C05497=1171.982,-20.083,-44.868,179.739,5.874,149.125
C05498=1171.976,-19.834,-44.881,179.742,5.874,149.124
C05499=1171.971,-19.584,-44.894,179.745,5.875,149.123
C05500=1171.966,-19.334,-44.907,179.746,5.875,149.123
C05501=1171.961,-19.085,-44.919,179.749,5.875,149.122
C05502=1171.956,-18.836,-44.932,179.751,5.876,149.122
C05503=1171.950,-18.586,-44.945,179.754,5.876,149.121
C05504=1171.946,-18.336,-44.958,179.756,5.877,149.120
C05505=1171.940,-18.086,-44.970,179.758,5.878,149.120
C05506=1171.935,-17.837,-44.983,179.761,5.878,149.119
C05507=1171.930,-17.588,-44.995,179.764,5.879,149.119
C05508=1171.925,-17.337,-45.009,179.766,5.879,149.118
C05509=1171.919,-17.088,-45.021,179.769,5.880,149.117
C05510=1171.914,-16.839,-45.034,179.771,5.880,149.117
C05511=1171.909,-16.589,-45.047,179.773,5.881,149.116
C05512=1171.904,-16.339,-45.060,179.776,5.882,149.116
C05513=1171.899,-16.090,-45.073,179.779,5.882,149.115
C05514=1171.894,-15.840,-45.085,179.781,5.883,149.114
C05515=1171.889,-15.590,-45.098,179.784,5.883,149.114
C05516=1171.883,-15.341,-45.112,179.785,5.883,149.113
C05517=1171.878,-15.091,-45.124,179.788,5.884,149.113
C05518=1171.874,-14.841,-45.137,179.791,5.884,149.112
C05519=1171.869,-14.592,-45.150,179.793,5.885,149.111
C05520=1171.863,-14.342,-45.163,179.795,5.886,149.111
C05521=1171.858,-14.092,-45.176,179.798,5.886,149.110
C05522=1171.853,-13.843,-45.189,179.800,5.887,149.110
C05523=1171.847,-13.593,-45.202,179.803,5.887,149.109
C05524=1171.842,-13.344,-45.214,179.806,5.888,149.108
C05525=1171.838,-13.094,-45.227,179.808,5.889,149.108
C05526=1171.832,-12.845,-45.240,179.810,5.889,149.107
C05527=1171.827,-12.595,-45.253,179.813,5.890,149.107
C05528=1171.822,-12.345,-45.266,179.815,5.890,149.106
C05529=1171.817,-12.096,-45.279,179.818,5.891,149.105
C05530=1171.812,-11.846,-45.293,179.820,5.892,149.105
C05531=1171.807,-11.597,-45.306,179.823,5.892,149.104
C05532=1171.801,-11.347,-45.319,179.825,5.892,149.103
C05533=1171.796,-11.097,-45.332,179.828,5.893,149.103
C05534=1171.791,-10.848,-45.344,179.830,5.894,149.102
C05535=1171.785,-10.598,-45.357,179.832,5.895,149.102
C05536=1171.781,-10.348,-45.370,179.835,5.895,149.101
C05537=1171.776,-10.099,-45.384,179.838,5.895,149.100
C05538=1171.771,-9.849,-45.397,179.840,5.896,149.100
C05539=1171.766,-9.600,-45.410,179.842,5.897,149.099
C05540=1171.760,-9.350,-45.423,179.845,5.897,149.098
C05541=1171.755,-9.100,-45.436,179.847,5.898,149.098
C05542=1171.750,-8.851,-45.449,179.850,5.898,149.097
C05543=1171.745,-8.601,-45.463,179.853,5.899,149.097
C05544=1171.740,-8.352,-45.476,179.855,5.900,149.096
C05545=1171.734,-8.102,-45.489,179.857,5.900,149.095
C05546=1171.730,-7.852,-45.502,179.860,5.901,149.095
C05547=1171.725,-7.604,-45.515,179.862,5.901,149.094
C05548=1171.720,-7.353,-45.529,179.864,5.901,149.094
C05549=1171.715,-7.104,-45.541,179.867,5.902,149.093
C05550=1171.709,-6.854,-45.554,179.869,5.902,149.092
C05551=1171.704,-6.605,-45.568,179.872,5.903,149.092
C05552=1171.699,-6.355,-45.581,179.874,5.904,149.091
C05553=1171.694,-6.105,-45.594,179.877,5.904,149.091
C05554=1171.689,-5.856,-45.608,179.879,5.905,149.090
C05555=1171.684,-5.606,-45.621,179.881,5.905,149.089
C05556=1171.678,-5.357,-45.634,179.884,5.906,149.089
C05557=1171.674,-5.106,-45.647,179.886,5.907,149.088
C05558=1171.668,-4.857,-45.661,179.889,5.907,149.088
C05559=1171.664,-4.607,-45.674,179.892,5.908,149.087
C05560=1171.658,-4.358,-45.687,179.894,5.908,149.086
C05561=1171.653,-4.109,-45.701,179.896,5.909,149.086
C05562=1171.648,-3.859,-45.714,179.900,5.910,149.085
C05563=1171.643,-3.610,-45.728,179.902,5.911,149.085
C05564=1171.638,-3.360,-45.741,179.905,5.911,149.084
C05565=1171.632,-3.110,-45.754,179.907,5.912,149.083
C05566=1171.627,-2.861,-45.768,179.909,5.913,149.083
C05567=1171.622,-2.611,-45.781,179.912,5.913,149.082
C05568=1171.617,-2.362,-45.795,179.914,5.914,149.082
C05569=1171.612,-2.112,-45.808,179.917,5.915,149.081
C05570=1171.607,-1.862,-45.821,179.920,5.915,149.080
C05571=1171.601,-1.613,-45.835,179.922,5.916,149.080
C05572=1171.597,-1.363,-45.848,179.924,5.916,149.079
C05573=1171.591,-1.114,-45.862,179.927,5.917,149.079
C05574=1171.586,-0.864,-45.875,179.929,5.918,149.078
C05575=1171.581,-0.615,-45.889,179.932,5.918,149.077
C05576=1171.576,-0.365,-45.902,179.934,5.919,149.077
C05577=1171.572,-0.115,-45.916,179.937,5.919,149.076
C05578=1171.566,0.134,-45.929,179.939,5.920,149.075
C05579=1171.561,0.384,-45.943,179.941,5.921,149.075
C05580=1171.556,0.633,-45.956,179.944,5.921,149.074
C05581=1171.551,0.883,-45.970,179.946,5.922,149.074
C05582=1171.545,1.133,-45.983,179.949,5.922,149.073
C05583=1171.541,1.382,-45.997,179.952,5.923,149.072
C05584=1171.535,1.632,-46.010,179.954,5.924,149.072
C05585=1171.530,1.901,-46.025,179.956,5.924,149.071
C05586=1171.524,2.171,-46.040,179.959,5.925,149.071
C05587=1171.519,2.440,-46.055,179.962,5.926,149.070
C05588=1171.513,2.708,-46.069,179.965,5.926,149.069
C05589=1171.508,2.959,-46.083,179.967,5.927,149.069
C05590=1171.503,3.208,-46.097,179.970,5.928,149.068
C05591=1171.498,3.458,-46.110,179.972,5.928,149.067
C05592=1171.493,3.707,-46.124,179.975,5.929,149.067
C05593=1171.488,3.956,-46.138,179.977,5.929,149.066
C05594=1171.483,4.206,-46.151,179.979,5.930,149.066
C05595=1171.478,4.456,-46.165,179.982,5.931,149.065
C05596=1171.473,4.705,-46.179,179.985,5.931,149.064
C05597=1171.467,4.956,-46.193,179.987,5.932,149.064
C05598=1171.462,5.204,-46.206,179.990,5.932,149.063
C05599=1171.457,5.454,-46.220,179.992,5.933,149.063
C05600=1171.452,5.704,-46.234,179.995,5.935,149.062
C05601=1171.447,5.953,-46.248,179.998,5.935,149.061
C05602=1171.442,6.203,-46.261,180.000,5.936,149.061
C05603=1171.437,6.453,-46.275,-179.998,5.936,149.060
C05604=1171.432,6.702,-46.289,-179.995,5.937,149.060
C05605=1171.427,6.952,-46.303,-179.993,5.938,149.059
C05606=1171.422,7.200,-46.317,-179.990,5.938,149.058
C05607=1171.417,7.451,-46.330,-179.988,5.939,149.058
C05608=1171.412,7.700,-46.344,-179.985,5.939,149.057
C05609=1171.406,7.949,-46.358,-179.983,5.940,149.057
C05610=1171.401,8.199,-46.373,-179.980,5.941,149.056
C05611=1171.397,8.449,-46.386,-179.978,5.941,149.055
C05612=1171.391,8.698,-46.399,-179.975,5.942,149.055
C05613=1171.386,8.948,-46.414,-179.973,5.942,149.054
C05614=1171.381,9.198,-46.428,-179.970,5.944,149.054
C05615=1171.376,9.447,-46.442,-179.968,5.945,149.053
C05616=1171.370,9.697,-46.455,-179.965,5.945,149.052
C05617=1171.365,9.947,-46.470,-179.962,5.946,149.052
C05618=1171.361,10.196,-46.483,-179.960,5.946,149.051
C05619=1171.356,10.445,-46.497,-179.957,5.947,149.051
C05620=1171.351,10.695,-46.512,-179.955,5.948,149.050
C05621=1171.346,10.945,-46.526,-179.953,5.948,149.049
C05622=1171.340,11.194,-46.539,-179.950,5.949,149.049
C05623=1171.335,11.444,-46.553,-179.948,5.949,149.048
C05624=1171.330,11.694,-46.568,-179.945,5.950,149.048
C05625=1171.325,11.943,-46.582,-179.942,5.951,149.047
C05626=1171.320,12.192,-46.595,-179.940,5.952,149.047
C05627=1171.315,12.442,-46.610,-179.937,5.953,149.046
C05628=1171.310,12.691,-46.624,-179.935,5.953,149.045
C05629=1171.305,12.941,-46.638,-179.932,5.954,149.045
C05630=1171.300,13.190,-46.652,-179.930,5.954,149.044
C05631=1171.295,13.440,-46.666,-179.927,5.955,149.044
C05632=1171.290,13.690,-46.681,-179.925,5.956,149.043
C05633=1171.285,13.939,-46.695,-179.923,5.956,149.042
C05634=1171.279,14.189,-46.708,-179.920,5.957,149.042
C05635=1171.274,14.439,-46.722,-179.917,5.958,149.041
C05636=1171.269,14.688,-46.737,-179.915,5.959,149.041
C05637=1171.264,14.938,-46.751,-179.912,5.960,149.040
C05638=1171.259,15.187,-46.765,-179.909,5.960,149.039
C05639=1171.254,15.437,-46.779,-179.907,5.961,149.039
C05640=1171.249,15.686,-46.793,-179.904,5.961,149.038
C05641=1171.244,15.936,-46.808,-179.902,5.962,149.038
C05642=1171.239,16.185,-46.823,-179.900,5.963,149.037
C05643=1171.233,16.434,-46.836,-179.896,5.964,149.036
C05644=1171.229,16.684,-46.851,-179.894,5.965,149.036
C05645=1171.224,16.934,-46.865,-179.892,5.965,149.035
C05646=1171.219,17.183,-46.879,-179.889,5.966,149.035
C05647=1171.214,17.433,-46.894,-179.887,5.967,149.034
C05648=1171.208,17.682,-46.908,-179.884,5.967,149.033
C05649=1171.203,17.932,-46.922,-179.882,5.968,149.033
C05650=1171.198,18.182,-46.936,-179.879,5.968,149.032
C05651=1171.193,18.431,-46.950,-179.877,5.970,149.032
C05652=1171.188,18.681,-46.965,-179.874,5.970,149.031
C05653=1171.184,18.930,-46.980,-179.871,5.971,149.030
C05654=1171.178,19.179,-46.994,-179.869,5.972,149.030
C05655=1171.173,19.429,-47.008,-179.866,5.972,149.029
C05656=1171.167,19.679,-47.023,-179.864,5.973,149.029
C05657=1171.162,19.928,-47.037,-179.862,5.974,149.028
C05658=1171.158,20.178,-47.051,-179.858,5.975,149.027
C05659=1171.153,20.427,-47.066,-179.856,5.976,149.027
C05660=1171.147,20.676,-47.080,-179.854,5.976,149.026
C05661=1171.142,20.926,-47.094,-179.851,5.977,149.026
C05662=1171.137,21.176,-47.109,-179.849,5.978,149.025
C05663=1171.132,21.425,-47.123,-179.846,5.978,149.024
C05664=1171.128,21.675,-47.138,-179.844,5.979,149.024
C05665=1171.122,21.925,-47.153,-179.841,5.980,149.023
C05666=1171.117,22.174,-47.167,-179.839,5.981,149.023
C05667=1171.112,22.424,-47.181,-179.836,5.981,149.022
C05668=1171.108,22.673,-47.196,-179.833,5.982,149.021
C05669=1171.102,22.922,-47.210,-179.831,5.983,149.021
C05670=1171.097,23.172,-47.225,-179.828,5.983,149.020
C05671=1171.091,23.422,-47.239,-179.826,5.985,149.020
C05672=1171.087,23.671,-47.254,-179.823,5.985,149.019
C05673=1171.082,23.921,-47.269,-179.820,5.986,149.019
C05674=1171.077,24.170,-47.283,-179.818,5.987,149.018
C05675=1171.072,24.419,-47.298,-179.816,5.987,149.017
C05676=1171.066,24.669,-47.313,-179.813,5.988,149.017
C05677=1171.062,24.919,-47.327,-179.810,5.989,149.016
C05678=1171.057,25.168,-47.342,-179.808,5.990,149.016
C05679=1171.052,25.418,-47.356,-179.805,5.991,149.015
C05680=1171.047,25.668,-47.371,-179.803,5.991,149.014
C05681=1171.042,25.917,-47.386,-179.801,5.992,149.014
C05682=1171.037,26.167,-47.401,-179.798,5.992,149.013
C05683=1171.032,26.416,-47.416,-179.795,5.994,149.013
C05684=1171.026,26.665,-47.429,-179.792,5.995,149.012
C05685=1171.021,26.915,-47.444,-179.790,5.995,149.012
C05686=1171.016,27.164,-47.459,-179.788,5.996,149.011
C05687=1171.011,27.414,-47.474,-179.785,5.996,149.010
C05688=1171.006,27.663,-47.489,-179.782,5.998,149.010
C05689=1171.001,27.932,-47.505,-179.780,5.999,149.009
C05690=1170.995,28.201,-47.521,-179.777,5.999,149.009
C05691=1170.990,28.470,-47.537,-179.774,6.000,149.008
C05692=1170.984,28.739,-47.553,-179.771,6.001,149.007
C05693=1170.980,28.988,-47.567,-179.769,6.002,149.007
C05694=1170.974,29.238,-47.582,-179.766,6.002,149.006
C05695=1170.969,29.487,-47.597,-179.764,6.004,149.006
C05696=1170.965,29.736,-47.612,-179.761,6.004,149.005
C05697=1170.959,29.986,-47.627,-179.758,6.005,149.004
C05698=1170.954,30.236,-47.642,-179.756,6.006,149.004
C05699=1170.949,30.486,-47.656,-179.753,6.006,149.003
C05700=1170.944,30.735,-47.671,-179.751,6.008,149.003
C05701=1170.939,30.984,-47.686,-179.748,6.008,149.002
C05702=1170.934,31.234,-47.701,-179.746,6.009,149.002
C05703=1170.929,31.483,-47.716,-179.743,6.010,149.001
C05704=1170.924,31.733,-47.731,-179.741,6.010,149.000
C05705=1170.919,31.982,-47.746,-179.738,6.012,149.000
C05706=1170.914,32.232,-47.761,-179.735,6.012,148.999
C05707=1170.909,32.482,-47.776,-179.733,6.013,148.999
C05708=1170.904,32.731,-47.791,-179.730,6.014,148.998
C05709=1170.899,32.981,-47.806,-179.728,6.015,148.998
C05710=1170.894,33.230,-47.821,-179.725,6.016,148.997
C05711=1170.889,33.480,-47.836,-179.722,6.016,148.996
C05712=1170.883,33.729,-47.851,-179.720,6.017,148.996
C05713=1170.879,33.978,-47.866,-179.718,6.018,148.995
C05714=1170.873,34.228,-47.881,-179.715,6.019,148.995
C05715=1170.868,34.477,-47.896,-179.712,6.020,148.994
C05716=1170.864,34.726,-47.911,-179.710,6.020,148.993
C05717=1170.858,34.976,-47.927,-179.707,6.021,148.993
C05718=1170.854,35.226,-47.941,-179.704,6.022,148.992
C05719=1170.849,35.476,-47.957,-179.702,6.023,148.992
C05720=1170.844,35.725,-47.972,-179.699,6.024,148.991
C05721=1170.838,35.975,-47.987,-179.697,6.025,148.991
C05722=1170.834,36.224,-48.002,-179.694,6.026,148.990
C05723=1170.828,36.473,-48.017,-179.691,6.026,148.989
C05724=1170.824,36.722,-48.032,-179.689,6.027,148.989
C05725=1170.818,36.972,-48.047,-179.687,6.028,148.988
C05726=1170.813,37.221,-48.062,-179.684,6.029,148.988
C05727=1170.809,37.472,-48.078,-179.681,6.030,148.987
C05728=1170.803,37.721,-48.094,-179.679,6.031,148.987
C05729=1170.798,37.970,-48.109,-179.676,6.031,148.986
C05730=1170.793,38.220,-48.124,-179.674,6.033,148.985
C05731=1170.788,38.469,-48.138,-179.671,6.033,148.985
C05732=1170.783,38.719,-48.154,-179.668,6.034,148.984
C05733=1170.779,38.968,-48.169,-179.666,6.035,148.984
C05734=1170.773,39.218,-48.185,-179.663,6.036,148.983
C05735=1170.768,39.467,-48.201,-179.661,6.037,148.982
C05736=1170.763,39.717,-48.215,-179.658,6.037,148.982
C05737=1170.758,39.966,-48.230,-179.656,6.038,148.981
C05738=1170.753,40.215,-48.245,-179.653,6.040,148.981
C05739=1170.748,40.465,-48.261,-179.650,6.040,148.980
C05740=1170.743,40.715,-48.277,-179.648,6.041,148.980
C05741=1170.738,40.964,-48.292,-179.645,6.041,148.979
C05742=1170.733,41.213,-48.308,-179.643,6.043,148.978
C05743=1170.728,41.462,-48.323,-179.640,6.044,148.978
C05744=1170.723,41.713,-48.339,-179.638,6.044,148.977
C05745=1170.718,41.962,-48.354,-179.635,6.045,148.977
C05746=1170.713,42.211,-48.369,-179.632,6.047,148.976
C05747=1170.708,42.460,-48.385,-179.630,6.047,148.976
C05748=1170.702,42.710,-48.400,-179.628,6.048,148.975
C05749=1170.698,42.960,-48.416,-179.624,6.049,148.974
C05750=1170.693,43.209,-48.431,-179.622,6.050,148.974
C05751=1170.688,43.458,-48.447,-179.620,6.051,148.973
C05752=1170.683,43.708,-48.462,-179.617,6.051,148.973
C05753=1170.678,43.958,-48.478,-179.614,6.053,148.972
C05754=1170.673,44.207,-48.493,-179.611,6.053,148.972
C05755=1170.667,44.456,-48.509,-179.609,6.054,148.971
C05756=1170.663,44.706,-48.524,-179.606,6.055,148.970
C05757=1170.658,44.956,-48.540,-179.604,6.056,148.970
C05758=1170.653,45.205,-48.555,-179.601,6.057,148.969
C05759=1170.648,45.454,-48.570,-179.599,6.057,148.969
C05760=1170.643,45.704,-48.586,-179.596,6.059,148.968
C05761=1170.638,45.954,-48.602,-179.593,6.059,148.968
C05762=1170.632,46.203,-48.618,-179.591,6.060,148.967
C05763=1170.628,46.452,-48.633,-179.588,6.062,148.966
C05764=1170.623,46.702,-48.649,-179.586,6.062,148.966
C05765=1170.618,46.951,-48.665,-179.583,6.063,148.965
C05766=1170.613,47.200,-48.680,-179.580,6.065,148.965
C05767=1170.608,47.450,-48.696,-179.578,6.065,148.964
C05768=1170.603,47.700,-48.711,-179.576,6.066,148.964
C05769=1170.598,47.949,-48.727,-179.572,6.067,148.963
C05770=1170.593,48.199,-48.743,-179.570,6.068,148.963
C05771=1170.588,48.448,-48.759,-179.568,6.069,148.962
C05772=1170.583,48.697,-48.774,-179.565,6.069,148.961
C05773=1170.578,48.947,-48.790,-179.562,6.071,148.961
C05774=1170.573,49.197,-48.806,-179.560,6.071,148.960
C05775=1170.568,49.446,-48.821,-179.557,6.072,148.960
C05776=1170.563,49.695,-48.838,-179.554,6.074,148.959
C05777=1170.558,49.945,-48.854,-179.552,6.074,148.959
C05778=1170.553,50.194,-48.869,-179.549,6.075,148.958
C05779=1170.548,50.444,-48.885,-179.547,6.077,148.958
C05780=1170.543,50.693,-48.901,-179.544,6.077,148.957
C05781=1170.538,50.942,-48.916,-179.542,6.078,148.956
C05782=1170.533,51.192,-48.932,-179.539,6.079,148.956
C05783=1170.528,51.441,-48.949,-179.536,6.080,148.955
C05784=1170.523,51.691,-48.965,-179.534,6.081,148.955
C05785=1170.518,51.941,-48.980,-179.531,6.082,148.954
C05786=1170.513,52.189,-48.996,-179.528,6.083,148.954
C05787=1170.509,52.439,-49.012,-179.526,6.084,148.953
C05788=1170.503,52.689,-49.028,-179.523,6.085,148.952
C05789=1170.499,52.938,-49.044,-179.520,6.085,148.952
C05790=1170.493,53.187,-49.060,-179.518,6.086,148.951
C05791=1170.488,53.437,-49.075,-179.515,6.088,148.951
C05792=1170.484,53.686,-49.092,-179.513,6.089,148.950
C05793=1170.478,53.955,-49.109,-179.510,6.090,148.950
C05794=1170.472,54.223,-49.126,-179.508,6.091,148.949
C05795=1170.467,54.492,-49.143,-179.504,6.092,148.948
C05796=1170.462,54.761,-49.160,-179.502,6.093,148.948
C05797=1170.457,55.010,-49.177,-179.499,6.094,148.947
C05798=1170.452,55.260,-49.193,-179.496,6.095,148.947
C05799=1170.447,55.509,-49.209,-179.494,6.096,148.946
C05800=1170.442,55.758,-49.225,-179.491,6.097,148.946
C05801=1170.437,56.008,-49.241,-179.489,6.098,148.945
C05802=1170.432,56.257,-49.257,-179.486,6.098,148.944
C05803=1170.427,56.506,-49.274,-179.483,6.100,148.944
C05804=1170.422,56.756,-49.289,-179.481,6.100,148.943
C05805=1170.417,57.005,-49.306,-179.478,6.101,148.943
C05806=1170.412,57.255,-49.321,-179.475,6.103,148.942
C05807=1170.408,57.504,-49.338,-179.473,6.103,148.942
C05808=1170.402,57.754,-49.354,-179.470,6.105,148.941
C05809=1170.398,58.003,-49.370,-179.467,6.105,148.940
C05810=1170.392,58.252,-49.386,-179.465,6.106,148.940
C05811=1170.387,58.502,-49.403,-179.462,6.108,148.939
C05812=1170.382,58.752,-49.419,-179.460,6.108,148.939
C05813=1170.377,59.001,-49.435,-179.457,6.109,148.938
C05814=1170.372,59.251,-49.451,-179.454,6.111,148.938
C05815=1170.367,59.500,-49.468,-179.452,6.111,148.937
C05816=1170.362,59.749,-49.484,-179.449,6.113,148.937
C05817=1170.357,59.999,-49.500,-179.446,6.113,148.936
C05818=1170.352,60.248,-49.516,-179.444,6.114,148.936
C05819=1170.348,60.497,-49.533,-179.441,6.115,148.935
C05820=1170.343,60.747,-49.548,-179.439,6.116,148.935
C05821=1170.337,60.996,-49.566,-179.436,6.118,148.934
C05822=1170.332,61.245,-49.582,-179.434,6.119,148.933
C05823=1170.327,61.495,-49.598,-179.431,6.119,148.933
C05824=1170.323,61.745,-49.615,-179.428,6.121,148.932
C05825=1170.318,61.994,-49.631,-179.426,6.122,148.932
C05826=1170.313,62.244,-49.647,-179.423,6.123,148.931
C05827=1170.307,62.493,-49.664,-179.421,6.124,148.931
C05828=1170.303,62.742,-49.681,-179.418,6.124,148.930
C05829=1170.297,62.992,-49.696,-179.415,6.126,148.930
C05830=1170.293,63.241,-49.713,-179.413,6.127,148.929
C05831=1170.288,63.490,-49.729,-179.410,6.128,148.929
C05832=1170.283,63.740,-49.746,-179.407,6.129,148.928
C05833=1170.278,63.990,-49.762,-179.405,6.130,148.928
C05834=1170.273,64.239,-49.779,-179.402,6.131,148.927
C05835=1170.268,64.488,-49.795,-179.400,6.132,148.926
C05836=1170.263,64.737,-49.812,-179.397,6.133,148.926
C05837=1170.258,64.987,-49.829,-179.394,6.134,148.925
C05838=1170.253,65.237,-49.845,-179.392,6.134,148.925
C05839=1170.248,65.486,-49.861,-179.389,6.136,148.924
C05840=1170.244,65.735,-49.878,-179.386,6.137,148.924
C05841=1170.238,65.985,-49.895,-179.384,6.138,148.923
C05842=1170.233,66.234,-49.911,-179.381,6.139,148.922
C05843=1170.229,66.483,-49.928,-179.378,6.141,148.922
C05844=1170.224,66.732,-49.944,-179.376,6.141,148.921
C05845=1170.218,66.982,-49.961,-179.374,6.142,148.921
C05846=1170.214,67.232,-49.978,-179.370,6.143,148.920
C05847=1170.209,67.481,-49.994,-179.368,6.144,148.920
C05848=1170.203,67.730,-50.011,-179.365,6.145,148.919
C05849=1170.199,67.980,-50.028,-179.363,6.146,148.919
C05850=1170.194,68.229,-50.044,-179.360,6.148,148.918
C05851=1170.189,68.478,-50.061,-179.357,6.149,148.918
C05852=1170.184,68.728,-50.078,-179.355,6.150,148.917
C05853=1170.179,68.977,-50.094,-179.352,6.151,148.917
C05854=1170.174,69.226,-50.112,-179.350,6.152,148.916
C05855=1170.169,69.476,-50.128,-179.347,6.153,148.915
C05856=1170.165,69.725,-50.145,-179.345,6.154,148.915
C05857=1170.159,69.975,-50.162,-179.341,6.155,148.914
C05858=1170.155,70.224,-50.178,-179.339,6.156,148.914
C05859=1170.150,70.473,-50.195,-179.336,6.157,148.913
C05860=1170.144,70.723,-50.212,-179.334,6.158,148.913
C05861=1170.140,70.972,-50.229,-179.331,6.160,148.912
C05862=1170.135,71.222,-50.246,-179.328,6.160,148.912
C05863=1170.130,71.471,-50.262,-179.326,6.162,148.911
C05864=1170.125,71.720,-50.279,-179.323,6.163,148.911
C05865=1170.120,71.970,-50.296,-179.321,6.164,148.910
C05866=1170.115,72.219,-50.313,-179.318,6.165,148.910
C05867=1170.110,72.468,-50.330,-179.316,6.166,148.909
C05868=1170.105,72.718,-50.346,-179.312,6.167,148.909
C05869=1170.100,72.968,-50.364,-179.310,6.168,148.908
C05870=1170.096,73.217,-50.381,-179.307,6.169,148.907
C05871=1170.090,73.466,-50.398,-179.305,6.170,148.907
C05872=1170.085,73.715,-50.415,-179.302,6.172,148.906
C05873=1170.080,73.965,-50.432,-179.299,6.172,148.906
C05874=1170.076,74.214,-50.449,-179.297,6.174,148.906
C05875=1170.070,74.464,-50.465,-179.294,6.175,148.905
C05876=1170.065,74.713,-50.482,-179.291,6.176,148.904
C05877=1170.060,74.962,-50.500,-179.289,6.177,148.904
C05878=1170.056,75.212,-50.517,-179.286,6.179,148.903
C05879=1170.051,75.462,-50.534,-179.283,6.179,148.903
C05880=1170.046,75.710,-50.550,-179.281,6.181,148.902
C05881=1170.041,75.959,-50.568,-179.278,6.181,148.902
C05882=1170.036,76.209,-50.585,-179.275,6.183,148.901
C05883=1170.031,76.459,-50.602,-179.273,6.184,148.901
C05884=1170.027,76.708,-50.619,-179.270,6.185,148.900
C05885=1170.021,76.957,-50.637,-179.268,6.186,148.900
C05886=1170.017,77.206,-50.653,-179.265,6.187,148.899
C05887=1170.011,77.456,-50.670,-179.262,6.188,148.899
C05888=1170.006,77.706,-50.688,-179.259,6.190,148.898
C05889=1170.002,77.955,-50.705,-179.257,6.190,148.897
C05890=1169.997,78.204,-50.722,-179.254,6.192,148.897
C05891=1169.992,78.453,-50.739,-179.252,6.193,148.896
C05892=1169.987,78.702,-50.757,-179.249,6.194,148.896
C05893=1169.982,78.952,-50.774,-179.246,6.195,148.895
C05894=1169.977,79.202,-50.791,-179.244,6.197,148.895
C05895=1169.972,79.451,-50.809,-179.241,6.197,148.894
C05896=1169.968,79.700,-50.825,-179.238,6.199,148.894
C05897=1169.962,79.969,-50.844,-179.236,6.199,148.893
C05898=1169.957,80.237,-50.863,-179.233,6.201,148.893
C05899=1169.951,80.506,-50.882,-179.230,6.202,148.892
C05900=1169.946,80.774,-50.899,-179.228,6.203,148.892
C05901=1169.941,81.023,-50.917,-179.224,6.205,148.891
C05902=1169.936,81.272,-50.935,-179.222,6.206,148.891
C05903=1169.931,81.522,-50.951,-179.219,6.207,148.890
C05904=1169.926,81.771,-50.969,-179.216,6.209,148.890
C05905=1169.921,82.021,-50.987,-179.214,6.209,148.889
C05906=1169.917,82.270,-51.004,-179.211,6.211,148.888
C05907=1169.912,82.520,-51.021,-179.209,6.212,148.888
C05908=1169.907,82.769,-51.039,-179.206,6.213,148.887
C05909=1169.902,83.019,-51.056,-179.203,6.214,148.887
C05910=1169.897,83.267,-51.074,-179.201,6.216,148.887
C05911=1169.892,83.517,-51.091,-179.198,6.216,148.886
C05912=1169.887,83.766,-51.109,-179.195,6.218,148.885
C05913=1169.882,84.015,-51.126,-179.193,6.218,148.885
C05914=1169.877,84.264,-51.143,-179.190,6.220,148.884
C05915=1169.873,84.514,-51.161,-179.187,6.221,148.884
C05916=1169.867,84.763,-51.179,-179.185,6.222,148.883
C05917=1169.862,85.013,-51.197,-179.182,6.224,148.883
C05918=1169.858,85.262,-51.213,-179.179,6.225,148.882
C05919=1169.853,85.511,-51.231,-179.177,6.226,148.882
C05920=1169.848,85.760,-51.249,-179.174,6.227,148.881
C05921=1169.843,86.010,-51.267,-179.171,6.228,148.881
C05922=1169.838,86.259,-51.284,-179.169,6.229,148.880
C05923=1169.833,86.509,-51.301,-179.166,6.231,148.880
C05924=1169.829,86.758,-51.319,-179.164,6.232,148.879
C05925=1169.824,87.007,-51.337,-179.161,6.233,148.879
C05926=1169.818,87.257,-51.354,-179.158,6.235,148.878
C05927=1169.814,87.506,-51.372,-179.156,6.235,148.878
C05928=1169.809,87.755,-51.390,-179.152,6.237,148.877
C05929=1169.804,88.005,-51.407,-179.150,6.238,148.877
C05930=1169.799,88.254,-51.425,-179.148,6.239,148.876
C05931=1169.794,88.503,-51.443,-179.145,6.240,148.876
C05932=1169.789,88.752,-51.461,-179.142,6.242,148.875
C05933=1169.784,89.002,-51.478,-179.139,6.243,148.875
C05934=1169.779,89.251,-51.496,-179.137,6.244,148.874
C05935=1169.774,89.500,-51.514,-179.134,6.246,148.874
C05936=1169.769,89.750,-51.532,-179.132,6.246,148.873
C05937=1169.764,89.999,-51.549,-179.129,6.248,148.873
C05938=1169.760,90.248,-51.567,-179.126,6.250,148.872
C05939=1169.755,90.497,-51.585,-179.123,6.250,148.872
C05940=1169.750,90.747,-51.603,-179.121,6.252,148.871
C05941=1169.745,90.996,-51.621,-179.118,6.252,148.870
C05942=1169.741,91.246,-51.638,-179.115,6.254,148.870
C05943=1169.736,91.495,-51.656,-179.113,6.255,148.870
C05944=1169.731,91.745,-51.674,-179.110,6.256,148.869
C05945=1169.726,91.994,-51.692,-179.107,6.258,148.869
C05946=1169.721,92.243,-51.710,-179.105,6.259,148.868
C05947=1169.716,92.492,-51.728,-179.102,6.260,148.868
C05948=1169.711,92.741,-51.746,-179.100,6.261,148.867
C05949=1169.706,92.991,-51.764,-179.097,6.263,148.867
C05950=1169.701,93.240,-51.782,-179.094,6.264,148.866
C05951=1169.696,93.490,-51.799,-179.092,6.265,148.866
C05952=1169.691,93.739,-51.817,-179.089,6.266,148.865
C05953=1169.687,93.989,-51.836,-179.086,6.267,148.865
C05954=1169.682,94.238,-51.854,-179.084,6.269,148.864
C05955=1169.677,94.487,-51.872,-179.081,6.270,148.864
C05956=1169.672,94.736,-51.890,-179.078,6.271,148.863
C05957=1169.667,94.985,-51.908,-179.076,6.273,148.863
C05958=1169.662,95.234,-51.926,-179.072,6.274,148.862
C05959=1169.658,95.484,-51.944,-179.070,6.275,148.862
C05960=1169.653,95.734,-51.962,-179.068,6.277,148.861
C05961=1169.648,95.983,-51.981,-179.065,6.277,148.861
C05962=1169.643,96.232,-51.999,-179.062,6.279,148.860
C05963=1169.638,96.481,-52.017,-179.060,6.281,148.860
C05964=1169.633,96.731,-52.035,-179.057,6.281,148.859
C05965=1169.628,96.980,-52.053,-179.054,6.283,148.859
C05966=1169.624,97.230,-52.071,-179.051,6.285,148.858
C05967=1169.619,97.479,-52.089,-179.049,6.285,148.858
C05968=1169.614,97.727,-52.108,-179.046,6.287,148.857
C05969=1169.609,97.976,-52.126,-179.044,6.288,148.857
C05970=1169.604,98.226,-52.144,-179.041,6.289,148.856
C05971=1169.599,98.475,-52.162,-179.038,6.291,148.856
C05972=1169.594,98.725,-52.180,-179.036,6.292,148.855
C05973=1169.589,98.974,-52.198,-179.033,6.293,148.855
C05974=1169.584,99.223,-52.216,-179.030,6.295,148.854
C05975=1169.580,99.473,-52.234,-179.028,6.296,148.854
C05976=1169.575,99.722,-52.254,-179.025,6.297,148.853
C05977=1169.570,99.971,-52.272,-179.022,6.299,148.853
C05978=1169.565,100.220,-52.290,-179.020,6.300,148.852
C05979=1169.560,100.470,-52.308,-179.017,6.301,148.852
C05980=1169.555,100.719,-52.326,-179.014,6.303,148.851
C05981=1169.550,100.968,-52.346,-179.012,6.304,148.851
C05982=1169.545,101.218,-52.364,-179.009,6.305,148.850
C05983=1169.541,101.467,-52.382,-179.006,6.307,148.850
C05984=1169.536,101.717,-52.400,-179.004,6.308,148.849
C05985=1169.532,101.965,-52.419,-179.001,6.309,148.849
C05986=1169.526,102.215,-52.437,-178.998,6.311,148.848
C05987=1169.521,102.464,-52.455,-178.996,6.312,148.848
C05988=1169.517,102.714,-52.474,-178.992,6.313,148.847
C05989=1169.511,102.963,-52.493,-178.990,6.315,148.847
C05990=1169.507,103.212,-52.511,-178.988,6.316,148.846
C05991=1169.502,103.461,-52.529,-178.985,6.317,148.846
C05992=1169.498,103.710,-52.548,-178.982,6.319,148.845
C05993=1169.492,103.960,-52.566,-178.980,6.320,148.845
C05994=1169.487,104.209,-52.584,-178.977,6.321,148.845
C05995=1169.483,104.458,-52.603,-178.974,6.323,148.844
C05996=1169.477,104.708,-52.622,-178.972,6.324,148.844
C05997=1169.473,104.956,-52.641,-178.969,6.325,148.843
C05998=1169.468,105.206,-52.659,-178.966,6.327,148.843
C05999=1169.463,105.456,-52.678,-178.963,6.328,148.842
C06000=1169.458,105.704,-52.696,-178.961,6.329,148.842
C06001=1169.452,105.973,-52.716,-178.958,6.331,148.841
C06002=1169.448,106.242,-52.736,-178.955,6.332,148.841
C06003=1169.442,106.510,-52.757,-178.952,6.334,148.840
C06004=1169.437,106.778,-52.776,-178.949,6.335,148.840
C06005=1169.433,107.027,-52.796,-178.947,6.336,148.839
C06006=1169.428,107.277,-52.814,-178.944,6.338,148.839
C06007=1169.423,107.525,-52.833,-178.941,6.339,148.838
C06008=1169.418,107.775,-52.851,-178.939,6.340,148.838
C06009=1169.413,108.024,-52.870,-178.936,6.342,148.837
C06010=1169.408,108.274,-52.889,-178.933,6.343,148.837
C06011=1169.404,108.523,-52.908,-178.930,6.345,148.836
C06012=1169.399,108.772,-52.926,-178.928,6.346,148.836
C06013=1169.394,109.021,-52.945,-178.925,6.347,148.835
C06014=1169.389,109.270,-52.963,-178.922,6.349,148.835
C06015=1169.384,109.519,-52.983,-178.920,6.350,148.834
C06016=1169.380,109.769,-53.001,-178.917,6.352,148.834
C06017=1169.374,110.018,-53.020,-178.914,6.353,148.833
C06018=1169.370,110.267,-53.039,-178.911,6.355,148.833
C06019=1169.365,110.517,-53.058,-178.909,6.356,148.833
C06020=1169.361,110.766,-53.077,-178.906,6.357,148.832
C06021=1169.355,111.015,-53.096,-178.903,6.359,148.832
C06022=1169.350,111.264,-53.114,-178.901,6.360,148.831
C06023=1169.346,111.514,-53.134,-178.898,6.361,148.831
C06024=1169.341,111.763,-53.152,-178.895,6.363,148.830
C06025=1169.336,112.012,-53.172,-178.892,6.365,148.830
C06026=1169.331,112.261,-53.190,-178.890,6.365,148.829
C06027=1169.327,112.511,-53.210,-178.888,6.367,148.829
C06028=1169.322,112.760,-53.228,-178.884,6.369,148.828
C06029=1169.317,113.009,-53.248,-178.882,6.370,148.828
C06030=1169.312,113.258,-53.267,-178.880,6.371,148.827
C06031=1169.307,113.507,-53.285,-178.877,6.373,148.827
C06032=1169.302,113.757,-53.305,-178.874,6.374,148.826
C06033=1169.297,114.005,-53.323,-178.871,6.376,148.826
C06034=1169.293,114.255,-53.343,-178.869,6.377,148.826
C06035=1169.287,114.505,-53.361,-178.866,6.379,148.825
C06036=1169.283,114.754,-53.381,-178.863,6.380,148.825
C06037=1169.278,115.003,-53.400,-178.860,6.382,148.824
C06038=1169.274,115.252,-53.419,-178.858,6.383,148.824
C06039=1169.268,115.501,-53.438,-178.855,6.384,148.823
C06040=1169.263,115.751,-53.457,-178.852,6.386,148.823
C06041=1169.259,116.000,-53.476,-178.849,6.387,148.822
C06042=1169.254,116.249,-53.495,-178.847,6.388,148.822
C06043=1169.248,116.498,-53.515,-178.845,6.390,148.821
C06044=1169.244,116.747,-53.534,-178.841,6.391,148.821
C06045=1169.240,116.997,-53.553,-178.839,6.393,148.820
C06046=1169.234,117.246,-53.573,-178.837,6.394,148.820
C06047=1169.230,117.495,-53.592,-178.834,6.396,148.820
C06048=1169.225,117.744,-53.610,-178.831,6.397,148.819
C06049=1169.220,117.994,-53.630,-178.828,6.399,148.819
C06050=1169.215,118.243,-53.649,-178.825,6.401,148.818
C06051=1169.211,118.492,-53.668,-178.823,6.401,148.818
C06052=1169.205,118.741,-53.688,-178.820,6.403,148.817
C06053=1169.201,118.991,-53.707,-178.817,6.405,148.817
C06054=1169.197,119.240,-53.726,-178.815,6.406,148.816
C06055=1169.191,119.489,-53.746,-178.812,6.407,148.816
C06056=1169.186,119.738,-53.765,-178.810,6.409,148.816
C06057=1169.181,119.987,-53.785,-178.807,6.410,148.815
C06058=1169.177,120.236,-53.804,-178.804,6.412,148.815
C06059=1169.172,120.486,-53.823,-178.801,6.414,148.814
C06060=1169.167,120.735,-53.843,-178.799,6.415,148.814
C06061=1169.162,120.984,-53.862,-178.796,6.416,148.813
C06062=1169.157,121.233,-53.882,-178.793,6.418,148.813
C06063=1169.153,121.482,-53.901,-178.790,6.419,148.812
C06064=1169.148,121.731,-53.921,-178.788,6.421,148.812
C06065=1169.143,121.980,-53.940,-178.786,6.422,148.811
C06066=1169.138,122.230,-53.960,-178.783,6.424,148.811
C06067=1169.134,122.479,-53.980,-178.780,6.425,148.810
C06068=1169.129,122.728,-53.998,-178.777,6.427,148.810
C06069=1169.124,122.978,-54.018,-178.774,6.429,148.810
C06070=1169.119,123.226,-54.037,-178.772,6.430,148.809
C06071=1169.114,123.476,-54.057,-178.769,6.431,148.809
C06072=1169.110,123.725,-54.077,-178.766,6.433,148.808
C06073=1169.104,123.974,-54.097,-178.763,6.434,148.808
C06074=1169.100,124.223,-54.116,-178.761,6.436,148.807
C06075=1169.096,124.473,-54.135,-178.759,6.437,148.807
C06076=1169.091,124.722,-54.155,-178.756,6.439,148.807
C06077=1169.086,124.970,-54.175,-178.753,6.440,148.806
C06078=1169.081,125.220,-54.195,-178.750,6.442,148.806
C06079=1169.076,125.470,-54.214,-178.747,6.444,148.805
C06080=1169.071,125.718,-54.234,-178.745,6.445,148.805
C06081=1169.067,125.967,-54.254,-178.742,6.446,148.804
C06082=1169.062,126.217,-54.274,-178.740,6.448,148.804
C06083=1169.057,126.466,-54.293,-178.737,6.449,148.803
C06084=1169.052,126.715,-54.313,-178.734,6.451,148.803
C06085=1169.047,126.964,-54.333,-178.731,6.453,148.803
C06086=1169.043,127.214,-54.353,-178.728,6.455,148.802
C06087=1169.037,127.463,-54.372,-178.726,6.455,148.802
C06088=1169.033,127.712,-54.392,-178.723,6.457,148.801
C06089=1169.028,127.961,-54.412,-178.720,6.459,148.801
C06090=1169.023,128.211,-54.432,-178.718,6.460,148.800
C06091=1169.018,128.459,-54.452,-178.715,6.462,148.800
C06092=1169.014,128.709,-54.471,-178.712,6.464,148.800
C06093=1169.009,128.958,-54.492,-178.710,6.466,148.799
C06094=1169.004,129.207,-54.511,-178.707,6.466,148.799
C06095=1168.999,129.456,-54.531,-178.704,6.468,148.798
C06096=1168.995,129.705,-54.551,-178.702,6.470,148.798
C06097=1168.990,129.955,-54.571,-178.699,6.471,148.797
C06098=1168.985,130.204,-54.591,-178.696,6.473,148.797
C06099=1168.980,130.452,-54.610,-178.693,6.475,148.797
C06100=1168.976,130.701,-54.631,-178.691,6.476,148.796
C06101=1168.971,130.951,-54.650,-178.688,6.477,148.796
C06102=1168.966,131.200,-54.671,-178.685,6.479,148.795
C06103=1168.962,131.449,-54.690,-178.683,6.480,148.795
C06104=1168.957,131.698,-54.710,-178.680,6.482,148.794
C06105=1168.951,131.967,-54.732,-178.677,6.484,148.794
C06106=1168.946,132.235,-54.753,-178.674,6.485,148.793
C06107=1168.941,132.504,-54.775,-178.671,6.487,148.793
C06108=1168.936,132.772,-54.797,-178.669,6.489,148.793
C06109=1168.931,133.022,-54.816,-178.666,6.491,148.792
C06110=1168.927,133.271,-54.837,-178.663,6.492,148.792
C06111=1168.921,133.520,-54.858,-178.660,6.494,148.791
C06112=1168.917,133.770,-54.877,-178.657,6.495,148.791
C06113=1168.912,134.019,-54.898,-178.655,6.497,148.790
C06114=1168.908,134.268,-54.917,-178.652,6.499,148.790
C06115=1168.903,134.516,-54.937,-178.649,6.501,148.790
C06116=1168.898,134.765,-54.958,-178.647,6.502,148.789
C06117=1168.893,135.015,-54.978,-178.645,6.503,148.789
C06118=1168.888,135.264,-54.998,-178.641,6.505,148.788
C06119=1168.884,135.513,-55.019,-178.639,6.506,148.788
C06120=1168.879,135.763,-55.038,-178.636,6.508,148.787
C06121=1168.874,136.012,-55.059,-178.633,6.510,148.787
C06122=1168.869,136.261,-55.080,-178.631,6.512,148.787
C06123=1168.865,136.510,-55.100,-178.628,6.513,148.786
C06124=1168.860,136.759,-55.119,-178.625,6.515,148.786
C06125=1168.854,137.008,-55.140,-178.622,6.517,148.786
C06126=1168.850,137.257,-55.161,-178.620,6.517,148.785
C06127=1168.845,137.507,-55.180,-178.617,6.519,148.785
C06128=1168.841,137.755,-55.201,-178.614,6.521,148.784
C06129=1168.836,138.005,-55.222,-178.612,6.523,148.784
C06130=1168.831,138.254,-55.242,-178.609,6.524,148.783
C06131=1168.827,138.503,-55.262,-178.606,6.526,148.783
C06132=1168.822,138.752,-55.282,-178.604,6.528,148.783
C06133=1168.817,139.001,-55.303,-178.601,6.530,148.782
C06134=1168.812,139.250,-55.323,-178.598,6.531,148.782
C06135=1168.808,139.499,-55.344,-178.596,6.533,148.781
C06136=1168.803,139.749,-55.365,-178.592,6.534,148.781
C06137=1168.798,139.998,-55.385,-178.590,6.536,148.780
C06138=1168.794,140.246,-55.405,-178.587,6.538,148.780
C06139=1168.788,140.496,-55.426,-178.585,6.539,148.780
C06140=1168.784,140.745,-55.446,-178.582,6.541,148.779
C06141=1168.779,140.995,-55.467,-178.579,6.542,148.779
C06142=1168.774,141.244,-55.487,-178.577,6.544,148.778
C06143=1168.770,141.492,-55.508,-178.574,6.546,148.778
C06144=1168.765,141.742,-55.529,-178.571,6.547,148.778
C06145=1168.760,141.991,-55.549,-178.569,6.549,148.777
C06146=1168.756,142.240,-55.569,-178.566,6.551,148.777
C06147=1168.751,142.489,-55.590,-178.563,6.553,148.777
C06148=1168.746,142.738,-55.611,-178.560,6.554,148.776
C06149=1168.741,142.987,-55.632,-178.557,6.556,148.776
C06150=1168.737,143.236,-55.652,-178.555,6.558,148.775
C06151=1168.732,143.485,-55.673,-178.552,6.559,148.775
C06152=1168.727,143.734,-55.693,-178.549,6.561,148.774
C06153=1168.722,143.984,-55.714,-178.547,6.563,148.774
C06154=1168.717,144.232,-55.735,-178.544,6.565,148.774
C06155=1168.713,144.481,-55.755,-178.541,6.566,148.773
C06156=1168.708,144.731,-55.776,-178.538,6.568,148.773
C06157=1168.703,144.980,-55.797,-178.536,6.570,148.772
C06158=1168.698,145.229,-55.817,-178.534,6.571,148.772
C06159=1168.694,145.477,-55.839,-178.531,6.572,148.772
C06160=1168.689,145.726,-55.860,-178.528,6.574,148.771
C06161=1168.684,145.975,-55.880,-178.526,6.576,148.771
C06162=1168.679,146.225,-55.901,-178.523,6.578,148.771
C06163=1168.675,146.474,-55.922,-178.520,6.579,148.770
C06164=1168.670,146.724,-55.943,-178.517,6.581,148.770
C06165=1168.665,146.973,-55.964,-178.514,6.583,148.769
C06166=1168.661,147.221,-55.985,-178.512,6.584,148.769
C06167=1168.656,147.470,-56.006,-178.509,6.586,148.768
C06168=1168.651,147.719,-56.026,-178.506,6.588,148.768
C06169=1168.646,147.969,-56.047,-178.503,6.590,148.768
C06170=1168.642,148.218,-56.067,-178.501,6.591,148.767
C06171=1168.637,148.466,-56.089,-178.498,6.593,148.767
C06172=1168.632,148.716,-56.110,-178.495,6.595,148.767
C06173=1168.628,148.965,-56.131,-178.493,6.596,148.766
C06174=1168.623,149.214,-56.152,-178.490,6.598,148.766
C06175=1168.618,149.463,-56.173,-178.487,6.600,148.765
C06176=1168.613,149.712,-56.194,-178.485,6.602,148.765
C06177=1168.608,149.961,-56.215,-178.482,6.603,148.765
C06178=1168.605,150.210,-56.236,-178.479,6.605,148.764
C06179=1168.600,150.460,-56.257,-178.476,6.607,148.764
C06180=1168.594,150.709,-56.278,-178.474,6.609,148.763
C06181=1168.590,150.957,-56.299,-178.471,6.610,148.763
C06182=1168.585,151.206,-56.320,-178.468,6.612,148.763
C06183=1168.580,151.456,-56.341,-178.466,6.614,148.762
C06184=1168.576,151.705,-56.363,-178.463,6.616,148.762
C06185=1168.571,151.954,-56.384,-178.460,6.617,148.762
C06186=1168.566,152.203,-56.405,-178.458,6.619,148.761
C06187=1168.561,152.452,-56.426,-178.455,6.621,148.761
C06188=1168.557,152.701,-56.447,-178.452,6.623,148.760
C06189=1168.552,152.950,-56.469,-178.450,6.624,148.760
C06190=1168.547,153.199,-56.490,-178.447,6.626,148.760
C06191=1168.542,153.448,-56.511,-178.444,6.628,148.759
C06192=1168.538,153.697,-56.532,-178.441,6.630,148.759
C06193=1168.533,153.946,-56.553,-178.439,6.631,148.759
C06194=1168.528,154.196,-56.575,-178.436,6.633,148.758
C06195=1168.524,154.444,-56.596,-178.433,6.635,148.758
C06196=1168.519,154.693,-56.617,-178.431,6.637,148.757
C06197=1168.514,154.942,-56.638,-178.427,6.639,148.757
C06198=1168.510,155.192,-56.660,-178.425,6.641,148.757
C06199=1168.505,155.440,-56.681,-178.422,6.643,148.756
C06200=1168.500,155.690,-56.702,-178.419,6.644,148.756
C06201=1168.495,155.939,-56.724,-178.417,6.646,148.756
C06202=1168.491,156.187,-56.745,-178.414,6.648,148.755
C06203=1168.486,156.437,-56.766,-178.411,6.650,148.755
C06204=1168.481,156.685,-56.788,-178.409,6.651,148.754
C06205=1168.477,156.935,-56.809,-178.406,6.653,148.754
C06206=1168.472,157.184,-56.831,-178.403,6.655,148.754
C06207=1168.467,157.432,-56.853,-178.400,6.657,148.753
C06208=1168.463,157.682,-56.874,-178.398,6.658,148.753
C06209=1168.457,157.950,-56.897,-178.395,6.660,148.753
C06210=1168.453,158.219,-56.920,-178.392,6.663,148.752
C06211=1168.447,158.489,-56.943,-178.389,6.665,148.752
C06212=1168.442,158.758,-56.966,-178.386,6.666,148.751
C06213=1168.438,159.007,-56.988,-178.384,6.668,148.751
C06214=1168.433,159.256,-57.010,-178.381,6.670,148.751
C06215=1168.428,159.504,-57.032,-178.378,6.672,148.750
C06216=1168.424,159.754,-57.053,-178.375,6.674,148.750
C06217=1168.419,160.003,-57.075,-178.372,6.676,148.750
C06218=1168.414,160.251,-57.096,-178.370,6.678,148.749
C06219=1168.410,160.501,-57.118,-178.367,6.679,148.749
C06220=1168.405,160.750,-57.139,-178.364,6.681,148.748
C06221=1168.400,160.999,-57.161,-178.362,6.683,148.748
C06222=1168.395,161.248,-57.183,-178.359,6.685,148.748
C06223=1168.391,161.497,-57.205,-178.356,6.686,148.747
C06224=1168.386,161.746,-57.227,-178.354,6.688,148.747
C06225=1168.381,161.995,-57.248,-178.351,6.690,148.747
C06226=1168.376,162.244,-57.269,-178.348,6.692,148.746
C06227=1168.372,162.493,-57.291,-178.345,6.693,148.746
C06228=1168.367,162.742,-57.313,-178.343,6.695,148.745
C06229=1168.363,162.991,-57.335,-178.340,6.698,148.745
C06230=1168.358,163.240,-57.357,-178.337,6.700,148.745
C06231=1168.353,163.489,-57.379,-178.335,6.702,148.745
C06232=1168.349,163.738,-57.401,-178.332,6.703,148.744
C06233=1168.344,163.987,-57.422,-178.329,6.705,148.744
C06234=1168.340,164.236,-57.444,-178.327,6.707,148.743
C06235=1168.335,164.485,-57.466,-178.324,6.709,148.743
C06236=1168.331,164.734,-57.488,-178.321,6.710,148.743
C06237=1168.326,164.982,-57.510,-178.318,6.712,148.742
C06238=1168.321,165.232,-57.532,-178.316,6.714,148.742
C06239=1168.316,165.481,-57.554,-178.313,6.716,148.742
C06240=1168.311,165.729,-57.576,-178.310,6.718,148.741
C06241=1168.307,165.979,-57.598,-178.307,6.720,148.741
C06242=1168.302,166.227,-57.619,-178.304,6.722,148.741
C06243=1168.298,166.477,-57.642,-178.302,6.724,148.740
C06244=1168.293,166.725,-57.663,-178.300,6.726,148.740
C06245=1168.288,166.975,-57.685,-178.297,6.727,148.740
C06246=1168.283,167.224,-57.708,-178.294,6.729,148.739
C06247=1168.279,167.473,-57.730,-178.291,6.732,148.739
C06248=1168.274,167.722,-57.751,-178.288,6.733,148.739
C06249=1168.269,167.971,-57.773,-178.286,6.735,148.738
C06250=1168.265,168.220,-57.795,-178.283,6.737,148.738
C06251=1168.260,168.469,-57.818,-178.280,6.739,148.737
C06252=1168.255,168.717,-57.840,-178.277,6.740,148.737
C06253=1168.251,168.967,-57.862,-178.275,6.742,148.737
C06254=1168.246,169.215,-57.884,-178.273,6.744,148.737
C06255=1168.241,169.465,-57.906,-178.269,6.747,148.736
C06256=1168.236,169.714,-57.928,-178.267,6.749,148.736
C06257=1168.232,169.962,-57.951,-178.264,6.750,148.735
C06258=1168.228,170.212,-57.973,-178.261,6.752,148.735
C06259=1168.222,170.461,-57.995,-178.259,6.754,148.735
C06260=1168.218,170.710,-58.017,-178.256,6.756,148.734
C06261=1168.213,170.959,-58.039,-178.254,6.758,148.734
C06262=1168.209,171.207,-58.062,-178.250,6.760,148.734
C06263=1168.203,171.456,-58.084,-178.248,6.762,148.734
C06264=1168.199,171.706,-58.106,-178.245,6.764,148.733
C06265=1168.195,171.954,-58.129,-178.242,6.766,148.733
C06266=1168.190,172.203,-58.151,-178.240,6.767,148.732
C06267=1168.185,172.453,-58.173,-178.237,6.769,148.732
C06268=1168.181,172.701,-58.195,-178.234,6.772,148.732
C06269=1168.176,172.950,-58.218,-178.232,6.774,148.732
C06270=1168.171,173.200,-58.240,-178.229,6.776,148.731
C06271=1168.167,173.448,-58.263,-178.226,6.777,148.731
C06272=1168.162,173.697,-58.285,-178.223,6.779,148.730
C06273=1168.157,173.946,-58.307,-178.221,6.781,148.730
C06274=1168.152,174.195,-58.330,-178.217,6.783,148.730
C06275=1168.148,174.444,-58.352,-178.215,6.785,148.730
C06276=1168.144,174.692,-58.375,-178.213,6.787,148.729
C06277=1168.139,174.942,-58.397,-178.210,6.789,148.729
C06278=1168.135,175.191,-58.420,-178.207,6.791,148.729
C06279=1168.129,175.440,-58.442,-178.205,6.793,148.728
C06280=1168.125,175.689,-58.464,-178.201,6.795,148.728
C06281=1168.121,175.938,-58.487,-178.199,6.797,148.727
C06282=1168.115,176.187,-58.509,-178.196,6.799,148.727
C06283=1168.111,176.435,-58.532,-178.194,6.801,148.727
C06284=1168.106,176.685,-58.555,-178.191,6.803,148.727
C06285=1168.102,176.933,-58.577,-178.188,6.805,148.726
C06286=1168.097,177.182,-58.601,-178.185,6.807,148.726
C06287=1168.093,177.431,-58.623,-178.182,6.809,148.726
C06288=1168.087,177.680,-58.646,-178.180,6.811,148.725
C06289=1168.083,177.929,-58.668,-178.178,6.812,148.725
C06290=1168.078,178.178,-58.691,-178.174,6.815,148.725
C06291=1168.073,178.427,-58.713,-178.172,6.817,148.724
C06292=1168.069,178.676,-58.736,-178.169,6.819,148.724
C06293=1168.065,178.925,-58.759,-178.167,6.821,148.724
C06294=1168.060,179.174,-58.782,-178.164,6.822,148.723
C06295=1168.055,179.422,-58.804,-178.161,6.825,148.723
C06296=1168.051,179.671,-58.827,-178.158,6.827,148.723
C06297=1168.046,179.921,-58.849,-178.155,6.829,148.722
C06298=1168.042,180.170,-58.873,-178.153,6.831,148.722
C06299=1168.037,180.418,-58.895,-178.150,6.833,148.722
C06300=1168.032,180.667,-58.918,-178.147,6.835,148.722
C06301=1168.027,180.916,-58.941,-178.145,6.837,148.721
C06302=1168.023,181.165,-58.964,-178.142,6.839,148.721
C06303=1168.018,181.413,-58.987,-178.140,6.841,148.721
C06304=1168.014,181.663,-59.009,-178.136,6.843,148.720
C06305=1168.009,181.912,-59.032,-178.134,6.845,148.720
C06306=1168.004,182.161,-59.056,-178.131,6.847,148.720
C06307=1168.000,182.410,-59.078,-178.128,6.849,148.719
C06308=1167.995,182.658,-59.101,-178.126,6.851,148.719
C06309=1167.990,182.907,-59.124,-178.123,6.853,148.719
C06310=1167.986,183.156,-59.147,-178.120,6.855,148.718
C06311=1167.981,183.405,-59.170,-178.118,6.857,148.718
C06312=1167.977,183.654,-59.194,-178.114,6.859,148.718
C06313=1167.972,183.924,-59.218,-178.112,6.861,148.718
C06314=1167.967,184.193,-59.243,-178.109,6.864,148.717
C06315=1167.962,184.463,-59.268,-178.106,6.866,148.717
C06316=1167.957,184.733,-59.292,-178.103,6.868,148.717
C06317=1167.952,184.982,-59.316,-178.100,6.870,148.716
C06318=1167.947,185.230,-59.339,-178.098,6.872,148.716
C06319=1167.943,185.479,-59.362,-178.095,6.874,148.716
C06320=1167.938,185.728,-59.385,-178.092,6.877,148.715
C06321=1167.934,185.977,-59.408,-178.089,6.878,148.715
C06322=1167.929,186.226,-59.432,-178.087,6.880,148.715
C06323=1167.925,186.475,-59.454,-178.084,6.882,148.714
C06324=1167.920,186.724,-59.478,-178.081,6.885,148.714
C06325=1167.916,186.973,-59.501,-178.079,6.887,148.714
C06326=1167.910,187.221,-59.524,-178.076,6.888,148.713
C06327=1167.906,187.470,-59.547,-178.073,6.890,148.713
C06328=1167.902,187.719,-59.570,-178.070,6.893,148.713
C06329=1167.897,187.968,-59.594,-178.068,6.895,148.713
C06330=1167.892,188.217,-59.617,-178.065,6.897,148.712
C06331=1167.887,188.466,-59.640,-178.062,6.900,148.712
C06332=1167.883,188.715,-59.664,-178.060,6.901,148.712
C06333=1167.878,188.964,-59.687,-178.057,6.903,148.711
C06334=1167.874,189.213,-59.710,-178.054,6.905,148.711
C06335=1167.869,189.462,-59.733,-178.051,6.908,148.711
C06336=1167.865,189.710,-59.757,-178.049,6.910,148.711
C06337=1167.860,189.958,-59.780,-178.046,6.911,148.710
C06338=1167.855,190.207,-59.804,-178.043,6.914,148.710
C06339=1167.850,190.456,-59.827,-178.041,6.916,148.710
C06340=1167.846,190.706,-59.850,-178.038,6.918,148.709
C06341=1167.841,190.955,-59.874,-178.035,6.920,148.709
C06342=1167.837,191.203,-59.898,-178.033,6.923,148.709
C06343=1167.833,191.452,-59.921,-178.030,6.924,148.709
C06344=1167.828,191.701,-59.944,-178.027,6.926,148.708
C06345=1167.823,191.950,-59.967,-178.024,6.929,148.708
C06346=1167.819,192.198,-59.991,-178.022,6.931,148.708
C06347=1167.814,192.447,-60.015,-178.019,6.933,148.707
C06348=1167.809,192.696,-60.038,-178.016,6.935,148.707
C06349=1167.805,192.945,-60.061,-178.014,6.937,148.707
C06350=1167.800,193.194,-60.085,-178.011,6.939,148.707
C06351=1167.796,193.443,-60.109,-178.008,6.941,148.706
C06352=1167.791,193.692,-60.132,-178.005,6.943,148.706
C06353=1167.786,193.940,-60.156,-178.003,6.945,148.706
C06354=1167.782,194.189,-60.180,-178.000,6.947,148.706
C06355=1167.777,194.438,-60.203,-177.997,6.950,148.705
C06356=1167.773,194.687,-60.227,-177.995,6.952,148.705
C06357=1167.768,194.936,-60.250,-177.992,6.954,148.705
C06358=1167.763,195.185,-60.274,-177.989,6.956,148.704
C06359=1167.759,195.433,-60.298,-177.987,6.958,148.704
C06360=1167.754,195.682,-60.321,-177.984,6.960,148.704
C06361=1167.750,195.931,-60.345,-177.981,6.963,148.704
C06362=1167.745,196.181,-60.370,-177.978,6.965,148.703
C06363=1167.741,196.429,-60.394,-177.976,6.967,148.703
C06364=1167.736,196.678,-60.417,-177.972,6.969,148.703
C06365=1167.731,196.927,-60.440,-177.970,6.971,148.703
C06366=1167.727,197.175,-60.464,-177.968,6.973,148.702
C06367=1167.722,197.425,-60.488,-177.964,6.976,148.702
C06368=1167.718,197.673,-60.512,-177.962,6.978,148.702
C06369=1167.713,197.922,-60.535,-177.959,6.980,148.701
C06370=1167.709,198.170,-60.559,-177.956,6.982,148.701
C06371=1167.703,198.419,-60.584,-177.954,6.984,148.701
C06372=1167.699,198.668,-60.607,-177.951,6.986,148.701
C06373=1167.695,198.917,-60.632,-177.948,6.989,148.700
C06374=1167.690,199.166,-60.655,-177.946,6.991,148.700
C06375=1167.686,199.415,-60.679,-177.943,6.993,148.700
C06376=1167.681,199.664,-60.703,-177.940,6.995,148.700
C06377=1167.676,199.912,-60.727,-177.938,6.997,148.699
C06378=1167.672,200.161,-60.751,-177.935,7.000,148.699
C06379=1167.667,200.410,-60.775,-177.932,7.002,148.699
C06380=1167.663,200.659,-60.799,-177.930,7.004,148.699
C06381=1167.659,200.907,-60.823,-177.926,7.006,148.698
C06382=1167.653,201.157,-60.847,-177.924,7.009,148.698
C06383=1167.649,201.405,-60.871,-177.922,7.010,148.698
C06384=1167.645,201.654,-60.895,-177.918,7.013,148.698
C06385=1167.640,201.903,-60.919,-177.916,7.015,148.697
C06386=1167.635,202.152,-60.944,-177.913,7.018,148.697
C06387=1167.631,202.400,-60.968,-177.910,7.019,148.697
C06388=1167.626,202.649,-60.992,-177.908,7.022,148.697
C06389=1167.622,202.898,-61.015,-177.905,7.024,148.696
C06390=1167.617,203.147,-61.040,-177.902,7.026,148.696
C06391=1167.613,203.396,-61.064,-177.900,7.028,148.696
C06392=1167.608,203.644,-61.088,-177.897,7.031,148.695
C06393=1167.603,203.893,-61.113,-177.894,7.033,148.695
C06394=1167.599,204.142,-61.136,-177.891,7.035,148.695
C06395=1167.595,204.391,-61.161,-177.888,7.037,148.695
C06396=1167.590,204.640,-61.186,-177.886,7.039,148.695
C06397=1167.585,204.888,-61.210,-177.883,7.042,148.694
C06398=1167.581,205.137,-61.234,-177.881,7.044,148.694
C06399=1167.576,205.385,-61.258,-177.878,7.047,148.694
C06400=1167.572,205.634,-61.283,-177.875,7.048,148.693
C06401=1167.567,205.883,-61.306,-177.873,7.050,148.693
C06402=1167.562,206.132,-61.331,-177.869,7.053,148.693
C06403=1167.558,206.381,-61.355,-177.867,7.055,148.693
C06404=1167.553,206.630,-61.380,-177.864,7.058,148.693
C06405=1167.549,206.878,-61.404,-177.862,7.060,148.692
C06406=1167.544,207.127,-61.429,-177.859,7.062,148.692
C06407=1167.540,207.376,-61.453,-177.856,7.064,148.692
C06408=1167.536,207.625,-61.477,-177.854,7.066,148.692
C06409=1167.530,207.873,-61.502,-177.850,7.069,148.691
C06410=1167.527,208.123,-61.526,-177.848,7.071,148.691
C06411=1167.521,208.371,-61.551,-177.846,7.073,148.691
C06412=1167.517,208.620,-61.575,-177.842,7.075,148.691
C06413=1167.512,208.868,-61.600,-177.840,7.078,148.690
C06414=1167.508,209.117,-61.624,-177.837,7.080,148.690
C06415=1167.503,209.366,-61.649,-177.835,7.082,148.690
C06416=1167.499,209.615,-61.673,-177.831,7.085,148.690
C06417=1167.494,209.885,-61.700,-177.829,7.087,148.689
C06418=1167.489,210.156,-61.727,-177.826,7.090,148.689
C06419=1167.484,210.427,-61.754,-177.823,7.092,148.689
C06420=1167.479,210.697,-61.780,-177.820,7.095,148.689
C06421=1167.474,210.945,-61.805,-177.817,7.097,148.689
C06422=1167.470,211.195,-61.830,-177.815,7.099,148.688
C06423=1167.465,211.443,-61.855,-177.812,7.102,148.688
C06424=1167.461,211.691,-61.879,-177.809,7.103,148.688
C06425=1167.457,211.940,-61.904,-177.806,7.106,148.688
C06426=1167.451,212.189,-61.929,-177.804,7.108,148.687
C06427=1167.448,212.438,-61.953,-177.801,7.111,148.687
C06428=1167.443,212.686,-61.979,-177.798,7.113,148.687
C06429=1167.438,212.935,-62.003,-177.796,7.116,148.687
C06430=1167.434,213.184,-62.028,-177.793,7.118,148.686
C06431=1167.429,213.433,-62.052,-177.790,7.119,148.686
C06432=1167.425,213.681,-62.077,-177.787,7.122,148.686
C06433=1167.420,213.930,-62.102,-177.785,7.124,148.686
C06434=1167.415,214.179,-62.127,-177.782,7.127,148.686
C06435=1167.412,214.427,-62.152,-177.779,7.129,148.685
C06436=1167.406,214.676,-62.177,-177.777,7.132,148.685
C06437=1167.402,214.926,-62.202,-177.774,7.134,148.685
C06438=1167.398,215.173,-62.226,-177.771,7.137,148.685
C06439=1167.393,215.423,-62.252,-177.769,7.138,148.684
C06440=1167.388,215.671,-62.276,-177.766,7.141,148.684
C06441=1167.385,215.920,-62.301,-177.763,7.143,148.684
C06442=1167.379,216.169,-62.326,-177.760,7.146,148.684
C06443=1167.375,216.417,-62.351,-177.758,7.148,148.684
C06444=1167.371,216.666,-62.376,-177.755,7.151,148.683
C06445=1167.366,216.915,-62.401,-177.752,7.152,148.683
C06446=1167.361,217.163,-62.426,-177.749,7.155,148.683
C06447=1167.356,217.412,-62.451,-177.747,7.157,148.683
C06448=1167.353,217.661,-62.476,-177.744,7.160,148.683
C06449=1167.348,217.909,-62.501,-177.741,7.162,148.682
C06450=1167.344,218.158,-62.527,-177.739,7.165,148.682
C06451=1167.338,218.407,-62.551,-177.736,7.167,148.682
C06452=1167.334,218.656,-62.577,-177.734,7.169,148.682
C06453=1167.330,218.905,-62.601,-177.730,7.171,148.681
C06454=1167.326,219.153,-62.627,-177.728,7.174,148.681
C06455=1167.321,219.402,-62.653,-177.725,7.176,148.681
C06456=1167.316,219.650,-62.677,-177.722,7.179,148.681
C06457=1167.312,219.899,-62.703,-177.720,7.181,148.681
C06458=1167.307,220.148,-62.728,-177.717,7.184,148.680
C06459=1167.303,220.396,-62.753,-177.714,7.186,148.680
C06460=1167.299,220.645,-62.778,-177.711,7.189,148.680
C06461=1167.294,220.894,-62.803,-177.709,7.191,148.680
C06462=1167.290,221.143,-62.829,-177.706,7.193,148.680
C06463=1167.285,221.391,-62.854,-177.704,7.195,148.679
C06464=1167.280,221.640,-62.879,-177.701,7.198,148.679
C06465=1167.276,221.888,-62.905,-177.698,7.200,148.679
C06466=1167.271,222.137,-62.930,-177.695,7.203,148.679
C06467=1167.267,222.386,-62.955,-177.693,7.205,148.679
C06468=1167.263,222.634,-62.980,-177.690,7.207,148.678
C06469=1167.259,222.883,-63.006,-177.687,7.210,148.678
C06470=1167.254,223.131,-63.031,-177.684,7.212,148.678
C06471=1167.249,223.381,-63.056,-177.682,7.214,148.678
C06472=1167.244,223.629,-63.082,-177.679,7.217,148.678
C06473=1167.240,223.878,-63.108,-177.677,7.219,148.677
C06474=1167.236,224.127,-63.133,-177.674,7.222,148.677
C06475=1167.231,224.375,-63.159,-177.671,7.224,148.677
C06476=1167.227,224.624,-63.184,-177.668,7.227,148.677
C06477=1167.222,224.873,-63.210,-177.665,7.229,148.677
C06478=1167.217,225.121,-63.235,-177.663,7.231,148.676
C06479=1167.213,225.370,-63.261,-177.660,7.234,148.676
C06480=1167.209,225.619,-63.286,-177.658,7.236,148.676
C06481=1167.204,225.867,-63.312,-177.655,7.239,148.676
C06482=1167.200,226.115,-63.338,-177.652,7.241,148.676
C06483=1167.196,226.364,-63.363,-177.649,7.244,148.676
C06484=1167.191,226.613,-63.388,-177.647,7.246,148.675
C06485=1167.186,226.862,-63.414,-177.644,7.249,148.675
C06486=1167.181,227.111,-63.440,-177.641,7.252,148.675
C06487=1167.177,227.359,-63.465,-177.639,7.253,148.675
C06488=1167.172,227.608,-63.491,-177.636,7.256,148.675
C06489=1167.168,227.857,-63.517,-177.633,7.258,148.674
C06490=1167.163,228.105,-63.542,-177.630,7.261,148.674
C06491=1167.159,228.354,-63.568,-177.628,7.263,148.674
C06492=1167.155,228.602,-63.594,-177.625,7.266,148.674
C06493=1167.151,228.851,-63.620,-177.622,7.269,148.674
C06494=1167.146,229.099,-63.645,-177.619,7.271,148.673
C06495=1167.141,229.348,-63.671,-177.617,7.273,148.673
C06496=1167.137,229.597,-63.698,-177.615,7.276,148.673
C06497=1167.133,229.845,-63.724,-177.611,7.278,148.673
C06498=1167.128,230.093,-63.749,-177.609,7.280,148.673
C06499=1167.124,230.342,-63.775,-177.606,7.283,148.673
C06500=1167.119,230.591,-63.800,-177.603,7.286,148.672
C06501=1167.114,230.840,-63.827,-177.601,7.288,148.672
C06502=1167.110,231.088,-63.852,-177.598,7.291,148.672
C06503=1167.105,231.337,-63.878,-177.595,7.293,148.672
C06504=1167.102,231.585,-63.904,-177.593,7.296,148.672
C06505=1167.097,231.834,-63.931,-177.589,7.298,148.672
C06506=1167.092,232.083,-63.956,-177.587,7.300,148.671
C06507=1167.088,232.331,-63.982,-177.585,7.303,148.671
C06508=1167.083,232.580,-64.008,-177.582,7.305,148.671
C06509=1167.079,232.829,-64.035,-177.579,7.308,148.671
C06510=1167.074,233.077,-64.060,-177.576,7.311,148.671
C06511=1167.070,233.326,-64.086,-177.574,7.313,148.671
C06512=1167.065,233.574,-64.112,-177.571,7.316,148.670
C06513=1167.061,233.823,-64.139,-177.569,7.318,148.670
C06514=1167.056,234.072,-64.164,-177.566,7.321,148.670
C06515=1167.052,234.320,-64.190,-177.563,7.324,148.670
C06516=1167.048,234.569,-64.217,-177.561,7.326,148.670
C06517=1167.043,234.818,-64.243,-177.557,7.328,148.670
C06518=1167.039,235.066,-64.268,-177.555,7.331,148.670
C06519=1167.034,235.314,-64.295,-177.552,7.333,148.669
C06520=1167.030,235.563,-64.321,-177.549,7.336,148.669
C06521=1167.025,235.834,-64.350,-177.546,7.339,148.669
C06522=1167.020,236.107,-64.379,-177.543,7.342,148.669
C06523=1167.015,236.378,-64.407,-177.540,7.344,148.669
C06524=1167.010,236.650,-64.436,-177.537,7.347,148.668
C06525=1167.006,236.898,-64.462,-177.535,7.349,148.668
C06526=1167.001,237.147,-64.489,-177.532,7.352,148.668
C06527=1166.997,237.396,-64.515,-177.529,7.355,148.668
C06528=1166.993,237.644,-64.541,-177.527,7.357,148.668
C06529=1166.988,237.893,-64.568,-177.524,7.360,148.668
C06530=1166.984,238.141,-64.593,-177.521,7.363,148.668
C06531=1166.979,238.390,-64.620,-177.519,7.365,148.667
C06532=1166.975,238.638,-64.646,-177.516,7.368,148.667
C06533=1166.970,238.887,-64.673,-177.514,7.370,148.667
C06534=1166.966,239.136,-64.699,-177.510,7.372,148.667
C06535=1166.961,239.384,-64.726,-177.508,7.375,148.667
C06536=1166.957,239.632,-64.753,-177.505,7.377,148.667
C06537=1166.952,239.881,-64.779,-177.503,7.380,148.667
C06538=1166.948,240.130,-64.805,-177.499,7.383,148.666
C06539=1166.943,240.379,-64.832,-177.497,7.385,148.666
C06540=1166.939,240.627,-64.858,-177.495,7.388,148.666
C06541=1166.935,240.875,-64.885,-177.492,7.391,148.666
C06542=1166.931,241.124,-64.911,-177.489,7.393,148.666
C06543=1166.926,241.373,-64.938,-177.486,7.396,148.666
C06544=1166.922,241.621,-64.965,-177.484,7.399,148.666
C06545=1166.917,241.870,-64.991,-177.481,7.401,148.666
C06546=1166.912,242.118,-65.018,-177.478,7.403,148.665
C06547=1166.908,242.367,-65.044,-177.475,7.406,148.665
C06548=1166.904,242.615,-65.071,-177.473,7.409,148.665
C06549=1166.900,242.864,-65.097,-177.470,7.412,148.665
C06550=1166.895,243.112,-65.124,-177.467,7.414,148.665
C06551=1166.890,243.361,-65.151,-177.465,7.416,148.665
C06552=1166.886,243.609,-65.178,-177.462,7.419,148.665
C06553=1166.881,243.858,-65.204,-177.460,7.422,148.664
C06554=1166.877,244.106,-65.231,-177.456,7.425,148.664
C06555=1166.873,244.355,-65.258,-177.454,7.427,148.664
C06556=1166.868,244.603,-65.285,-177.451,7.430,148.664
C06557=1166.864,244.852,-65.311,-177.449,7.433,148.664
C06558=1166.860,245.100,-65.338,-177.446,7.435,148.664
C06559=1166.855,245.349,-65.365,-177.443,7.438,148.664
C06560=1166.851,245.597,-65.391,-177.440,7.441,148.663
C06561=1166.846,245.846,-65.418,-177.438,7.443,148.663
C06562=1166.842,246.095,-65.446,-177.435,7.446,148.663
C06563=1166.837,246.344,-65.473,-177.432,7.448,148.663
C06564=1166.833,246.592,-65.499,-177.429,7.451,148.663
C06565=1166.829,246.840,-65.526,-177.427,7.453,148.663
C06566=1166.824,247.089,-65.553,-177.425,7.456,148.663
C06567=1166.819,247.337,-65.580,-177.422,7.459,148.663
C06568=1166.815,247.585,-65.607,-177.419,7.461,148.662
C06569=1166.811,247.834,-65.634,-177.416,7.464,148.662
C06570=1166.806,248.082,-65.661,-177.414,7.467,148.662
C06571=1166.802,248.331,-65.688,-177.411,7.469,148.662
C06572=1166.797,248.580,-65.715,-177.409,7.472,148.662
C06573=1166.794,248.828,-65.742,-177.406,7.475,148.662
C06574=1166.789,249.077,-65.769,-177.403,7.478,148.662
C06575=1166.784,249.325,-65.796,-177.401,7.480,148.662
C06576=1166.780,249.574,-65.823,-177.398,7.483,148.662
C06577=1166.775,249.822,-65.851,-177.395,7.486,148.662
C06578=1166.772,250.071,-65.878,-177.392,7.489,148.661
C06579=1166.767,250.319,-65.905,-177.390,7.490,148.661
C06580=1166.763,250.568,-65.932,-177.387,7.493,148.661
C06581=1166.758,250.816,-65.959,-177.384,7.496,148.661
C06582=1166.753,251.065,-65.986,-177.382,7.498,148.661
C06583=1166.749,251.313,-66.013,-177.379,7.501,148.661
C06584=1166.745,251.562,-66.041,-177.376,7.504,148.661
C06585=1166.740,251.810,-66.068,-177.374,7.507,148.661
C06586=1166.736,252.059,-66.095,-177.371,7.509,148.660
C06587=1166.732,252.307,-66.122,-177.368,7.512,148.660
C06588=1166.727,252.555,-66.149,-177.365,7.515,148.660
C06589=1166.723,252.804,-66.177,-177.363,7.518,148.660
C06590=1166.719,253.052,-66.204,-177.360,7.520,148.660
C06591=1166.714,253.301,-66.231,-177.358,7.523,148.660
C06592=1166.710,253.549,-66.259,-177.355,7.526,148.660
C06593=1166.705,253.798,-66.286,-177.352,7.529,148.660
C06594=1166.701,254.046,-66.313,-177.350,7.531,148.660
C06595=1166.696,254.294,-66.341,-177.347,7.534,148.660
C06596=1166.692,254.543,-66.368,-177.344,7.537,148.660
C06597=1166.688,254.792,-66.395,-177.341,7.540,148.659
C06598=1166.683,255.040,-66.423,-177.339,7.542,148.659
C06599=1166.679,255.288,-66.450,-177.336,7.545,148.659
C06600=1166.674,255.536,-66.478,-177.334,7.548,148.659
C06601=1166.670,255.785,-66.506,-177.331,7.551,148.659
C06602=1166.666,256.034,-66.533,-177.328,7.554,148.659
C06603=1166.661,256.282,-66.560,-177.325,7.555,148.659
C06604=1166.657,256.531,-66.588,-177.323,7.558,148.659
C06605=1166.653,256.779,-66.616,-177.320,7.561,148.659
C06606=1166.648,257.028,-66.643,-177.317,7.564,148.659
C06607=1166.644,257.276,-66.671,-177.315,7.566,148.659
C06608=1166.639,257.525,-66.698,-177.312,7.569,148.658
C06609=1166.635,257.773,-66.726,-177.309,7.572,148.658
C06610=1166.631,258.022,-66.754,-177.307,7.575,148.658
C06611=1166.626,258.270,-66.781,-177.304,7.578,148.658
C06612=1166.622,258.518,-66.809,-177.302,7.580,148.658
C06613=1166.618,258.767,-66.837,-177.299,7.583,148.658
C06614=1166.614,259.015,-66.864,-177.296,7.586,148.658
C06615=1166.608,259.263,-66.892,-177.293,7.589,148.658
C06616=1166.604,259.512,-66.920,-177.290,7.592,148.658
C06617=1166.600,259.760,-66.948,-177.288,7.594,148.658
C06618=1166.595,260.008,-66.975,-177.285,7.597,148.658
C06619=1166.592,260.257,-67.003,-177.283,7.600,148.658
C06620=1166.586,260.506,-67.031,-177.280,7.603,148.658
C06621=1166.583,260.754,-67.059,-177.278,7.605,148.657
C06622=1166.578,261.002,-67.087,-177.275,7.608,148.657
C06623=1166.574,261.250,-67.115,-177.272,7.611,148.657
C06624=1166.570,261.499,-67.142,-177.269,7.614,148.657
C06625=1166.565,261.773,-67.173,-177.267,7.617,148.657
C06626=1166.560,262.045,-67.203,-177.264,7.620,148.657
C06627=1166.555,262.318,-67.235,-177.261,7.623,148.657
C06628=1166.550,262.592,-67.266,-177.258,7.627,148.657
C06629=1166.545,262.840,-67.293,-177.255,7.628,148.657
C06630=1166.542,263.089,-67.321,-177.252,7.631,148.657
C06631=1166.537,263.337,-67.349,-177.250,7.634,148.657
C06632=1166.533,263.585,-67.377,-177.247,7.637,148.657
C06633=1166.529,263.833,-67.405,-177.244,7.640,148.657
C06634=1166.525,264.082,-67.433,-177.241,7.643,148.656
C06635=1166.519,264.331,-67.461,-177.239,7.645,148.656
C06636=1166.515,264.579,-67.489,-177.236,7.648,148.656
C06637=1166.511,264.827,-67.517,-177.234,7.651,148.656
C06638=1166.506,265.075,-67.545,-177.231,7.654,148.656
C06639=1166.502,265.324,-67.573,-177.228,7.657,148.656
C06640=1166.497,265.572,-67.602,-177.225,7.660,148.656
C06641=1166.494,265.821,-67.630,-177.223,7.662,148.656
C06642=1166.489,266.069,-67.658,-177.220,7.665,148.656
C06643=1166.485,266.317,-67.686,-177.218,7.668,148.656
C06644=1166.480,266.565,-67.714,-177.215,7.671,148.656
C06645=1166.476,266.814,-67.743,-177.212,7.674,148.656
C06646=1166.472,267.062,-67.771,-177.210,7.677,148.656
C06647=1166.468,267.311,-67.799,-177.208,7.680,148.656
C06648=1166.463,267.559,-67.827,-177.205,7.683,148.656
C06649=1166.459,267.807,-67.855,-177.202,7.685,148.656
C06650=1166.454,268.056,-67.884,-177.199,7.688,148.656
C06651=1166.450,268.304,-67.912,-177.197,7.691,148.656
C06652=1166.446,268.553,-67.941,-177.194,7.694,148.656
C06653=1166.441,268.801,-67.968,-177.192,7.697,148.656
C06654=1166.437,269.050,-67.997,-177.189,7.699,148.655
C06655=1166.432,269.298,-68.025,-177.186,7.702,148.655
C06656=1166.428,269.546,-68.054,-177.184,7.705,148.655
C06657=1166.424,269.794,-68.082,-177.181,7.708,148.655
C06658=1166.419,270.043,-68.111,-177.178,7.711,148.655
C06659=1166.416,270.291,-68.139,-177.175,7.714,148.655
C06660=1166.411,270.540,-68.167,-177.173,7.716,148.655
C06661=1166.407,270.788,-68.195,-177.170,7.719,148.655
C06662=1166.402,271.036,-68.225,-177.168,7.722,148.655
C06663=1166.398,271.285,-68.253,-177.165,7.725,148.655
C06664=1166.394,271.533,-68.281,-177.162,7.728,148.655
C06665=1166.389,271.781,-68.310,-177.159,7.731,148.655
C06666=1166.385,272.029,-68.339,-177.157,7.735,148.655
C06667=1166.380,272.277,-68.367,-177.154,7.737,148.655
C06668=1166.376,272.526,-68.396,-177.152,7.740,148.655
C06669=1166.372,272.774,-68.425,-177.149,7.743,148.655
C06670=1166.367,273.023,-68.453,-177.147,7.746,148.655
C06671=1166.363,273.271,-68.481,-177.144,7.749,148.655
C06672=1166.359,273.519,-68.511,-177.141,7.751,148.655
C06673=1166.354,273.768,-68.539,-177.138,7.754,148.655
C06674=1166.350,274.016,-68.567,-177.136,7.757,148.655
C06675=1166.346,274.264,-68.597,-177.133,7.760,148.655
C06676=1166.341,274.513,-68.625,-177.131,7.762,148.655
C06677=1166.338,274.761,-68.654,-177.128,7.766,148.655
C06678=1166.333,275.009,-68.683,-177.126,7.769,148.655
C06679=1166.328,275.258,-68.711,-177.123,7.772,148.655
C06680=1166.325,275.506,-68.740,-177.120,7.775,148.655
C06681=1166.320,275.754,-68.769,-177.117,7.778,148.655
C06682=1166.316,276.003,-68.798,-177.115,7.781,148.654
C06683=1166.311,276.251,-68.826,-177.112,7.784,148.654
C06684=1166.308,276.499,-68.855,-177.109,7.787,148.654
C06685=1166.303,276.748,-68.884,-177.107,7.789,148.655
C06686=1166.298,276.995,-68.913,-177.105,7.792,148.654
C06687=1166.294,277.244,-68.942,-177.102,7.795,148.654
C06688=1166.290,277.492,-68.971,-177.099,7.798,148.654
C06689=1166.286,277.740,-69.000,-177.096,7.801,148.654
C06690=1166.281,277.989,-69.028,-177.094,7.804,148.654
C06691=1166.277,278.237,-69.058,-177.091,7.807,148.654
C06692=1166.272,278.486,-69.087,-177.089,7.810,148.654
C06693=1166.269,278.734,-69.116,-177.086,7.813,148.654
C06694=1166.264,278.981,-69.145,-177.083,7.816,148.654
C06695=1166.260,279.230,-69.173,-177.081,7.818,148.654
C06696=1166.255,279.478,-69.203,-177.078,7.821,148.654
C06697=1166.251,279.727,-69.232,-177.075,7.824,148.654
C06698=1166.247,279.976,-69.261,-177.073,7.827,148.654
C06699=1166.243,280.223,-69.289,-177.070,7.830,148.654
C06700=1166.239,280.471,-69.319,-177.068,7.833,148.654
C06701=1166.234,280.719,-69.348,-177.065,7.836,148.654
C06702=1166.230,280.968,-69.377,-177.062,7.839,148.654
C06703=1166.226,281.217,-69.407,-177.059,7.842,148.654
C06704=1166.221,281.464,-69.436,-177.057,7.845,148.654
C06705=1166.217,281.712,-69.465,-177.054,7.848,148.654
C06706=1166.213,281.961,-69.495,-177.052,7.851,148.654
C06707=1166.208,282.210,-69.523,-177.049,7.854,148.654
C06708=1166.204,282.458,-69.553,-177.047,7.857,148.654
C06709=1166.200,282.706,-69.582,-177.044,7.859,148.654
C06710=1166.195,282.954,-69.611,-177.042,7.863,148.654
C06711=1166.191,283.202,-69.641,-177.039,7.866,148.654
C06712=1166.187,283.450,-69.670,-177.036,7.869,148.654
C06713=1166.182,283.699,-69.699,-177.033,7.872,148.654
C06714=1166.178,283.947,-69.728,-177.031,7.875,148.654
C06715=1166.174,284.196,-69.758,-177.028,7.878,148.654
C06716=1166.170,284.444,-69.787,-177.026,7.881,148.654
C06717=1166.165,284.692,-69.817,-177.023,7.884,148.654
C06718=1166.161,284.940,-69.846,-177.020,7.887,148.654
C06719=1166.156,285.188,-69.875,-177.018,7.890,148.654
C06720=1166.152,285.436,-69.905,-177.015,7.893,148.654
C06721=1166.148,285.684,-69.934,-177.012,7.896,148.654
C06722=1166.144,285.933,-69.964,-177.010,7.899,148.654
C06723=1166.140,286.181,-69.993,-177.007,7.902,148.654
C06724=1166.136,286.429,-70.023,-177.005,7.905,148.654
C06725=1166.131,286.678,-70.052,-177.002,7.907,148.654
C06726=1166.127,286.926,-70.081,-177.000,7.910,148.654
C06727=1166.122,287.174,-70.112,-176.997,7.913,148.654
C06728=1166.118,287.423,-70.141,-176.995,7.917,148.654
C06729=1166.113,287.697,-70.174,-176.991,7.920,148.654
C06730=1166.109,287.972,-70.206,-176.988,7.923,148.654
C06731=1166.104,288.247,-70.239,-176.985,7.927,148.654
C06732=1166.099,288.522,-70.272,-176.982,7.930,148.654
C06733=1166.095,288.770,-70.302,-176.980,7.933,148.654
C06734=1166.091,289.018,-70.331,-176.977,7.936,148.654
C06735=1166.086,289.266,-70.362,-176.975,7.939,148.654
C06736=1166.082,289.515,-70.391,-176.972,7.942,148.654
C06737=1166.078,289.763,-70.420,-176.970,7.946,148.655
C06738=1166.074,290.011,-70.451,-176.967,7.949,148.654
C06739=1166.070,290.259,-70.480,-176.964,7.952,148.654
C06740=1166.065,290.507,-70.510,-176.961,7.955,148.654
C06741=1166.061,290.756,-70.540,-176.959,7.958,148.655
C06742=1166.057,291.003,-70.570,-176.956,7.961,148.655
C06743=1166.052,291.252,-70.599,-176.954,7.964,148.655
C06744=1166.048,291.500,-70.629,-176.951,7.967,148.655
C06745=1166.044,291.748,-70.659,-176.949,7.970,148.655
C06746=1166.039,291.996,-70.689,-176.946,7.973,148.655
C06747=1166.035,292.244,-70.718,-176.943,7.976,148.655
C06748=1166.031,292.492,-70.749,-176.941,7.979,148.655
C06749=1166.027,292.741,-70.779,-176.938,7.982,148.655
C06750=1166.023,292.989,-70.809,-176.935,7.985,148.655
C06751=1166.018,293.238,-70.839,-176.934,7.988,148.655
C06752=1166.014,293.486,-70.869,-176.931,7.991,148.655
C06753=1166.010,293.733,-70.899,-176.928,7.994,148.655
C06754=1166.005,293.982,-70.929,-176.926,7.997,148.655
C06755=1166.001,294.230,-70.959,-176.923,8.000,148.655
C06756=1165.997,294.478,-70.988,-176.920,8.003,148.655
C06757=1165.993,294.726,-71.019,-176.918,8.006,148.655
C06758=1165.988,294.974,-71.049,-176.915,8.009,148.655
C06759=1165.984,295.222,-71.079,-176.912,8.012,148.655
C06760=1165.980,295.471,-71.109,-176.910,8.015,148.655
C06761=1165.976,295.719,-71.139,-176.907,8.018,148.655
C06762=1165.972,295.967,-71.169,-176.905,8.021,148.655
C06763=1165.968,296.215,-71.200,-176.902,8.025,148.655
C06764=1165.963,296.464,-71.230,-176.900,8.028,148.655
C06765=1165.959,296.711,-71.260,-176.897,8.030,148.655
C06766=1165.955,296.959,-71.290,-176.895,8.034,148.655
C06767=1165.951,297.208,-71.320,-176.891,8.038,148.655
C06768=1165.947,297.456,-71.351,-176.889,8.041,148.655
C06769=1165.942,297.704,-71.381,-176.886,8.044,148.656
C06770=1165.938,297.952,-71.411,-176.883,8.047,148.656
C06771=1165.933,298.200,-71.442,-176.881,8.050,148.656
C06772=1165.929,298.448,-71.472,-176.878,8.053,148.656
C06773=1165.925,298.697,-71.502,-176.876,8.056,148.656
C06774=1165.921,298.945,-71.532,-176.873,8.059,148.656
C06775=1165.917,299.193,-71.563,-176.871,8.062,148.656
C06776=1165.913,299.440,-71.593,-176.868,8.065,148.656
C06777=1165.908,299.689,-71.623,-176.866,8.069,148.656
C06778=1165.904,299.937,-71.654,-176.863,8.072,148.656
C06779=1165.900,300.185,-71.685,-176.860,8.074,148.656
C06780=1165.895,300.433,-71.715,-176.858,8.078,148.656
C06781=1165.891,300.681,-71.745,-176.855,8.081,148.656
C06782=1165.887,300.929,-71.776,-176.853,8.084,148.656
C06783=1165.883,301.178,-71.806,-176.850,8.087,148.656
C06784=1165.879,301.426,-71.837,-176.847,8.090,148.656
C06785=1165.874,301.673,-71.868,-176.845,8.093,148.656
C06786=1165.870,301.921,-71.898,-176.842,8.096,148.656
C06787=1165.866,302.170,-71.929,-176.840,8.100,148.657
C06788=1165.862,302.418,-71.960,-176.837,8.103,148.657
C06789=1165.857,302.666,-71.989,-176.834,8.105,148.657
C06790=1165.853,302.914,-72.020,-176.832,8.109,148.657
C06791=1165.849,303.163,-72.051,-176.829,8.112,148.657
C06792=1165.845,303.410,-72.081,-176.827,8.115,148.657
C06793=1165.840,303.658,-72.112,-176.824,8.118,148.657
C06794=1165.836,303.907,-72.143,-176.822,8.121,148.657
C06795=1165.832,304.155,-72.173,-176.819,8.124,148.657
C06796=1165.828,304.403,-72.204,-176.817,8.127,148.657
C06797=1165.823,304.650,-72.235,-176.814,8.131,148.657
C06798=1165.819,304.899,-72.266,-176.811,8.134,148.657
C06799=1165.815,305.147,-72.296,-176.809,8.138,148.657
C06800=1165.811,305.395,-72.327,-176.806,8.141,148.657
C06801=1165.807,305.643,-72.358,-176.804,8.144,148.658
C06802=1165.802,305.891,-72.389,-176.801,8.147,148.658
C06803=1165.798,306.139,-72.420,-176.799,8.150,148.658
C06804=1165.794,306.387,-72.451,-176.796,8.153,148.658
C06805=1165.790,306.635,-72.482,-176.793,8.156,148.658
C06806=1165.785,306.883,-72.512,-176.791,8.159,148.658
C06807=1165.781,307.132,-72.543,-176.788,8.162,148.658
C06808=1165.777,307.380,-72.574,-176.786,8.166,148.658
C06809=1165.774,307.627,-72.605,-176.783,8.169,148.658
C06810=1165.769,307.875,-72.636,-176.781,8.172,148.658
C06811=1165.764,308.123,-72.667,-176.778,8.175,148.658
C06812=1165.760,308.372,-72.698,-176.776,8.178,148.658
C06813=1165.756,308.619,-72.730,-176.773,8.181,148.658
C06814=1165.751,308.867,-72.760,-176.770,8.185,148.659
C06815=1165.747,309.116,-72.791,-176.767,8.188,148.659
C06816=1165.744,309.363,-72.822,-176.765,8.192,148.659
C06817=1165.740,309.612,-72.853,-176.762,8.194,148.659
C06818=1165.735,309.859,-72.884,-176.760,8.198,148.659
C06819=1165.731,310.107,-72.915,-176.757,8.201,148.659
C06820=1165.727,310.355,-72.947,-176.755,8.204,148.659
C06821=1165.722,310.603,-72.978,-176.752,8.207,148.659
C06822=1165.718,310.852,-73.009,-176.750,8.210,148.659
C06823=1165.714,311.099,-73.040,-176.747,8.213,148.659
C06824=1165.710,311.348,-73.071,-176.745,8.217,148.659
C06825=1165.705,311.596,-73.102,-176.742,8.220,148.659
C06826=1165.702,311.844,-73.134,-176.739,8.224,148.660
C06827=1165.697,312.092,-73.165,-176.737,8.227,148.660
C06828=1165.693,312.340,-73.197,-176.734,8.230,148.660
C06829=1165.689,312.588,-73.227,-176.732,8.233,148.660
C06830=1165.684,312.835,-73.259,-176.729,8.236,148.660
C06831=1165.680,313.084,-73.290,-176.727,8.239,148.660
C06832=1165.676,313.331,-73.321,-176.724,8.242,148.660
C06833=1165.672,313.610,-73.356,-176.721,8.246,148.660
C06834=1165.667,313.886,-73.391,-176.719,8.250,148.660
C06835=1165.662,314.163,-73.426,-176.715,8.253,148.660
C06836=1165.658,314.440,-73.462,-176.713,8.257,148.661
C06837=1165.653,314.688,-73.493,-176.710,8.260,148.661
C06838=1165.650,314.936,-73.524,-176.707,8.264,148.661
C06839=1165.645,315.184,-73.556,-176.705,8.267,148.661
C06840=1165.641,315.432,-73.587,-176.702,8.270,148.661
C06841=1165.637,315.680,-73.618,-176.700,8.273,148.661
C06842=1165.633,315.928,-73.650,-176.697,8.276,148.661
C06843=1165.628,316.176,-73.682,-176.695,8.280,148.661
C06844=1165.624,316.424,-73.714,-176.692,8.283,148.661
C06845=1165.620,316.671,-73.745,-176.690,8.286,148.661
C06846=1165.616,316.920,-73.776,-176.687,8.290,148.662
C06847=1165.612,317.168,-73.808,-176.684,8.293,148.662
C06848=1165.608,317.415,-73.839,-176.682,8.296,148.662
C06849=1165.604,317.664,-73.871,-176.679,8.299,148.662
C06850=1165.599,317.912,-73.903,-176.677,8.302,148.662
C06851=1165.595,318.160,-73.935,-176.675,8.306,148.662
C06852=1165.592,318.408,-73.966,-176.672,8.309,148.662
C06853=1165.587,318.655,-73.998,-176.670,8.312,148.662
C06854=1165.583,318.904,-74.029,-176.666,8.316,148.662
C06855=1165.578,319.151,-74.061,-176.664,8.319,148.663
C06856=1165.575,319.399,-74.093,-176.662,8.322,148.663
C06857=1165.571,319.648,-74.125,-176.659,8.325,148.663
C06858=1165.566,319.895,-74.156,-176.657,8.329,148.663
C06859=1165.562,320.143,-74.189,-176.654,8.332,148.663
C06860=1165.558,320.392,-74.220,-176.652,8.335,148.663
C06861=1165.554,320.639,-74.251,-176.650,8.338,148.663
C06862=1165.550,320.887,-74.283,-176.646,8.342,148.663
C06863=1165.546,321.136,-74.316,-176.644,8.345,148.664
C06864=1165.541,321.383,-74.347,-176.642,8.349,148.664
C06865=1165.538,321.631,-74.379,-176.639,8.352,148.664
C06866=1165.533,321.879,-74.411,-176.637,8.355,148.664
C06867=1165.529,322.127,-74.443,-176.634,8.358,148.664
C06868=1165.525,322.375,-74.475,-176.632,8.361,148.664
C06869=1165.521,322.623,-74.507,-176.629,8.365,148.664
C06870=1165.516,322.870,-74.539,-176.626,8.369,148.665
C06871=1165.513,323.118,-74.570,-176.624,8.372,148.665
C06872=1165.508,323.367,-74.603,-176.621,8.375,148.665
C06873=1165.504,323.614,-74.634,-176.619,8.378,148.665
C06874=1165.500,323.862,-74.666,-176.616,8.381,148.665
C06875=1165.496,324.110,-74.699,-176.613,8.385,148.665
C06876=1165.492,324.358,-74.731,-176.611,8.388,148.665
C06877=1165.487,324.606,-74.763,-176.608,8.391,148.665
C06878=1165.484,324.854,-74.795,-176.606,8.395,148.666
C06879=1165.480,325.102,-74.827,-176.604,8.398,148.666
C06880=1165.475,325.350,-74.859,-176.601,8.401,148.666
C06881=1165.471,325.597,-74.891,-176.598,8.405,148.666
C06882=1165.467,325.845,-74.924,-176.596,8.408,148.666
C06883=1165.463,326.093,-74.956,-176.594,8.412,148.667
C06884=1165.459,326.341,-74.988,-176.591,8.415,148.667
C06885=1165.455,326.589,-75.020,-176.589,8.418,148.667
C06886=1165.450,326.837,-75.053,-176.586,8.421,148.667
C06887=1165.447,327.085,-75.085,-176.583,8.425,148.667
C06888=1165.442,327.333,-75.117,-176.581,8.428,148.667
C06889=1165.439,327.581,-75.149,-176.578,8.432,148.667
C06890=1165.434,327.828,-75.182,-176.576,8.435,148.668
C06891=1165.430,328.076,-75.214,-176.573,8.438,148.668
C06892=1165.426,328.324,-75.246,-176.571,8.441,148.668
C06893=1165.422,328.572,-75.279,-176.568,8.445,148.668
C06894=1165.418,328.820,-75.311,-176.566,8.449,148.668
C06895=1165.414,329.067,-75.343,-176.563,8.452,148.668
C06896=1165.409,329.315,-75.376,-176.561,8.455,148.668
C06897=1165.405,329.564,-75.408,-176.559,8.458,148.669
C06898=1165.402,329.811,-75.441,-176.556,8.462,148.669
C06899=1165.397,330.059,-75.473,-176.553,8.465,148.669
C06900=1165.394,330.307,-75.506,-176.551,8.469,148.669
C06901=1165.389,330.555,-75.538,-176.548,8.472,148.669
C06902=1165.384,330.803,-75.570,-176.546,8.475,148.669
C06903=1165.381,331.050,-75.603,-176.543,8.479,148.669
C06904=1165.376,331.298,-75.635,-176.541,8.482,148.670
C06905=1165.372,331.546,-75.668,-176.538,8.486,148.670
C06906=1165.369,331.794,-75.700,-176.536,8.489,148.670
C06907=1165.364,332.042,-75.733,-176.534,8.492,148.670
C06908=1165.360,332.290,-75.767,-176.530,8.496,148.670
C06909=1165.357,332.538,-75.798,-176.528,8.499,148.671
C06910=1165.352,332.785,-75.831,-176.526,8.502,148.671
C06911=1165.347,333.033,-75.864,-176.523,8.506,148.671
C06912=1165.343,333.281,-75.897,-176.521,8.509,148.671
C06913=1165.340,333.528,-75.929,-176.518,8.513,148.671
C06914=1165.335,333.777,-75.962,-176.516,8.516,148.671
C06915=1165.331,334.024,-75.995,-176.513,8.519,148.672
C06916=1165.328,334.272,-76.028,-176.511,8.523,148.672
C06917=1165.323,334.520,-76.060,-176.508,8.527,148.672
C06918=1165.319,334.768,-76.093,-176.506,8.530,148.672
C06919=1165.315,335.016,-76.126,-176.503,8.533,148.672
C06920=1165.311,335.264,-76.159,-176.501,8.536,148.672
C06921=1165.307,335.511,-76.191,-176.499,8.540,148.673
C06922=1165.303,335.759,-76.224,-176.496,8.544,148.673
C06923=1165.299,336.007,-76.258,-176.493,8.547,148.673
C06924=1165.295,336.255,-76.290,-176.491,8.550,148.673
C06925=1165.290,336.503,-76.323,-176.489,8.554,148.674
C06926=1165.287,336.750,-76.356,-176.485,8.558,148.674
C06927=1165.283,336.998,-76.389,-176.483,8.561,148.674
C06928=1165.279,337.246,-76.422,-176.481,8.564,148.674
C06929=1165.274,337.494,-76.455,-176.479,8.567,148.674
C06930=1165.270,337.742,-76.488,-176.476,8.572,148.674
C06931=1165.266,337.990,-76.521,-176.473,8.575,148.675
C06932=1165.262,338.237,-76.554,-176.471,8.578,148.675
C06933=1165.258,338.485,-76.587,-176.469,8.581,148.675
C06934=1165.254,338.732,-76.620,-176.466,8.585,148.675
C06935=1165.250,338.980,-76.653,-176.463,8.588,148.675
C06936=1165.246,339.228,-76.686,-176.461,8.592,148.676
C06937=1165.241,339.507,-76.724,-176.458,8.596,148.676
C06938=1165.237,339.787,-76.761,-176.455,8.600,148.676
C06939=1165.232,340.067,-76.798,-176.453,8.603,148.676
C06940=1165.227,340.347,-76.835,-176.450,8.607,148.676
C06941=1165.223,340.595,-76.869,-176.448,8.611,148.677
C06942=1165.219,340.842,-76.902,-176.445,8.615,148.677
C06943=1165.215,341.090,-76.935,-176.443,8.618,148.677
C06944=1165.211,341.338,-76.968,-176.440,8.621,148.677
C06945=1165.207,341.585,-77.002,-176.437,8.626,148.678
C06946=1165.203,341.833,-77.035,-176.435,8.629,148.678
C06947=1165.199,342.080,-77.068,-176.433,8.632,148.678
C06948=1165.195,342.328,-77.101,-176.431,8.635,148.678
C06949=1165.190,342.576,-77.135,-176.428,8.639,148.679
C06950=1165.186,342.824,-77.168,-176.425,8.643,148.679
C06951=1165.182,343.071,-77.201,-176.423,8.646,148.679
C06952=1165.179,343.320,-77.234,-176.421,8.649,148.679
C06953=1165.174,343.567,-77.269,-176.418,8.653,148.679
C06954=1165.170,343.815,-77.302,-176.416,8.657,148.680
C06955=1165.166,344.063,-77.335,-176.413,8.660,148.680
C06956=1165.162,344.310,-77.368,-176.410,8.664,148.680
C06957=1165.158,344.557,-77.402,-176.408,8.667,148.680
C06958=1165.154,344.805,-77.435,-176.406,8.671,148.680
C06959=1165.150,345.054,-77.469,-176.404,8.674,148.681
C06960=1165.146,345.301,-77.502,-176.401,8.678,148.681
C06961=1165.141,345.549,-77.536,-176.398,8.681,148.681
C06962=1165.137,345.796,-77.570,-176.396,8.685,148.681
C06963=1165.133,346.044,-77.603,-176.393,8.689,148.682
C06964=1165.129,346.291,-77.637,-176.391,8.692,148.682
C06965=1165.126,346.540,-77.670,-176.389,8.695,148.682
C06966=1165.122,346.787,-77.703,-176.386,8.700,148.682
C06967=1165.117,347.035,-77.738,-176.383,8.703,148.683
C06968=1165.113,347.283,-77.771,-176.381,8.706,148.683
C06969=1165.109,347.530,-77.804,-176.378,8.710,148.683
C06970=1165.106,347.778,-77.838,-176.376,8.714,148.683
C06971=1165.101,348.026,-77.872,-176.374,8.717,148.683
C06972=1165.097,348.273,-77.906,-176.372,8.720,148.684
C06973=1165.093,348.521,-77.939,-176.369,8.725,148.684
C06974=1165.089,348.768,-77.973,-176.367,8.728,148.684
C06975=1165.085,349.017,-78.007,-176.364,8.731,148.685
C06976=1165.081,349.264,-78.041,-176.362,8.735,148.685
C06977=1165.077,349.512,-78.074,-176.359,8.739,148.685
C06978=1165.072,349.759,-78.109,-176.357,8.742,148.685
C06979=1165.069,350.008,-78.142,-176.354,8.746,148.685
C06980=1165.065,350.255,-78.176,-176.352,8.749,148.686
C06981=1165.061,350.502,-78.209,-176.350,8.753,148.686
C06982=1165.057,350.751,-78.244,-176.347,8.757,148.686
C06983=1165.053,350.998,-78.278,-176.345,8.760,148.687
C06984=1165.048,351.246,-78.312,-176.342,8.764,148.687
C06985=1165.044,351.493,-78.346,-176.340,8.768,148.687
C06986=1165.041,351.741,-78.380,-176.337,8.771,148.687
C06987=1165.036,351.989,-78.413,-176.335,8.775,148.688
C06988=1165.032,352.236,-78.447,-176.333,8.779,148.688
C06989=1165.029,352.484,-78.482,-176.330,8.782,148.688
C06990=1165.024,352.732,-78.515,-176.328,8.785,148.688
C06991=1165.020,352.979,-78.549,-176.325,8.789,148.689
C06992=1165.016,353.227,-78.584,-176.323,8.793,148.689
C06993=1165.012,353.475,-78.617,-176.320,8.797,148.689
C06994=1165.008,353.722,-78.651,-176.318,8.800,148.690
C06995=1165.004,353.970,-78.686,-176.316,8.804,148.690
C06996=1165.000,354.217,-78.720,-176.313,8.808,148.690
C06997=1164.996,354.464,-78.754,-176.311,8.811,148.690
C06998=1164.992,354.713,-78.788,-176.309,8.815,148.691
C06999=1164.988,354.960,-78.822,-176.306,8.819,148.691
C07000=1164.985,355.208,-78.856,-176.304,8.822,148.691
C07001=1164.980,355.455,-78.891,-176.302,8.826,148.692
C07002=1164.976,355.702,-78.925,-176.299,8.830,148.692
C07003=1164.972,355.951,-78.960,-176.297,8.833,148.692
C07004=1164.968,356.198,-78.994,-176.294,8.837,148.692
C07005=1164.964,356.446,-79.028,-176.292,8.841,148.693
C07006=1164.960,356.694,-79.062,-176.290,8.844,148.693
C07007=1164.956,356.941,-79.096,-176.287,8.848,148.693
C07008=1164.952,357.189,-79.130,-176.284,8.852,148.693
C07009=1164.948,357.436,-79.165,-176.283,8.855,148.694
C07010=1164.944,357.684,-79.200,-176.280,8.859,148.694
C07011=1164.940,357.931,-79.233,-176.277,8.863,148.694
C07012=1164.936,358.180,-79.268,-176.275,8.867,148.695
C07013=1164.932,358.427,-79.302,-176.273,8.870,148.695
C07014=1164.928,358.674,-79.337,-176.270,8.874,148.695
C07015=1164.924,358.922,-79.372,-176.268,8.878,148.696
C07016=1164.920,359.169,-79.406,-176.266,8.881,148.696
C07017=1164.916,359.417,-79.441,-176.263,8.885,148.696
C07018=1164.912,359.664,-79.475,-176.261,8.889,148.697
C07019=1164.908,359.912,-79.510,-176.258,8.893,148.697
C07020=1164.904,360.159,-79.544,-176.256,8.896,148.697
C07021=1164.901,360.407,-79.578,-176.254,8.900,148.698
C07022=1164.896,360.655,-79.613,-176.251,8.904,148.698
C07023=1164.892,360.902,-79.648,-176.249,8.908,148.698
C07024=1164.889,361.149,-79.682,-176.246,8.912,148.699
C07025=1164.885,361.397,-79.717,-176.244,8.915,148.699
C07026=1164.880,361.645,-79.751,-176.242,8.920,148.699
C07027=1164.876,361.893,-79.786,-176.239,8.923,148.699
C07028=1164.873,362.139,-79.821,-176.237,8.926,148.700
C07029=1164.869,362.388,-79.856,-176.235,8.931,148.700
C07030=1164.865,362.636,-79.890,-176.233,8.934,148.701
C07031=1164.861,362.883,-79.924,-176.230,8.938,148.701
C07032=1164.857,363.130,-79.960,-176.228,8.942,148.701
C07033=1164.852,363.378,-79.994,-176.226,8.946,148.702
C07034=1164.849,363.626,-80.029,-176.223,8.950,148.702
C07035=1164.845,363.872,-80.064,-176.221,8.953,148.702
C07036=1164.841,364.120,-80.099,-176.218,8.957,148.703
C07037=1164.837,364.369,-80.133,-176.217,8.961,148.703
C07038=1164.833,364.615,-80.169,-176.214,8.965,148.704
C07039=1164.829,364.864,-80.203,-176.212,8.969,148.704
C07040=1164.825,365.110,-80.238,-176.210,8.972,148.704
C07041=1164.820,365.393,-80.278,-176.208,8.977,148.705
C07042=1164.816,365.676,-80.318,-176.205,8.981,148.705
C07043=1164.811,365.958,-80.357,-176.202,8.985,148.705
C07044=1164.807,366.240,-80.397,-176.200,8.990,148.706
C07045=1164.803,366.488,-80.433,-176.197,8.994,148.706
C07046=1164.799,366.735,-80.467,-176.196,8.998,148.707
C07047=1164.795,366.983,-80.503,-176.194,9.001,148.707
C07048=1164.791,367.230,-80.537,-176.191,9.005,148.708
C07049=1164.787,367.478,-80.573,-176.189,9.009,148.708
C07050=1164.783,367.726,-80.608,-176.187,9.012,148.708
C07051=1164.779,367.973,-80.643,-176.185,9.017,148.709
C07052=1164.775,368.220,-80.678,-176.183,9.021,148.709
C07053=1164.771,368.468,-80.713,-176.181,9.024,148.710
C07054=1164.768,368.715,-80.748,-176.178,9.029,148.710
C07055=1164.764,368.963,-80.783,-176.177,9.032,148.711
C07056=1164.760,369.210,-80.818,-176.175,9.036,148.711
C07057=1164.756,369.457,-80.853,-176.173,9.039,148.711
C07058=1164.752,369.705,-80.888,-176.170,9.044,148.712
C07059=1164.748,369.953,-80.924,-176.169,9.047,148.712
C07060=1164.744,370.200,-80.959,-176.167,9.051,148.713
C07061=1164.740,370.448,-80.994,-176.165,9.055,148.713
C07062=1164.736,370.695,-81.029,-176.163,9.059,148.714
C07063=1164.733,370.943,-81.065,-176.161,9.063,148.714
C07064=1164.728,371.189,-81.100,-176.159,9.066,148.715
C07065=1164.724,371.438,-81.135,-176.158,9.070,148.715
C07066=1164.720,371.685,-81.171,-176.156,9.074,148.716
C07067=1164.716,371.932,-81.206,-176.153,9.078,148.716
C07068=1164.712,372.180,-81.242,-176.152,9.082,148.717
C07069=1164.708,372.428,-81.277,-176.150,9.086,148.717
C07070=1164.704,372.675,-81.312,-176.148,9.090,148.718
C07071=1164.700,372.922,-81.347,-176.147,9.093,148.718
C07072=1164.696,373.170,-81.383,-176.145,9.097,148.719
C07073=1164.693,373.417,-81.418,-176.144,9.101,148.719
C07074=1164.689,373.665,-81.454,-176.142,9.105,148.720
C07075=1164.685,373.911,-81.489,-176.140,9.108,148.720
C07076=1164.681,374.160,-81.524,-176.138,9.112,148.721
C07077=1164.676,374.407,-81.560,-176.137,9.116,148.722
C07078=1164.673,374.655,-81.596,-176.136,9.120,148.722
C07079=1164.669,374.902,-81.631,-176.134,9.123,148.723
C07080=1164.665,375.149,-81.666,-176.132,9.127,148.723
C07081=1164.661,375.397,-81.702,-176.131,9.131,148.724
C07082=1164.658,375.644,-81.737,-176.129,9.135,148.724
C07083=1164.654,375.892,-81.773,-176.128,9.139,148.725
C07084=1164.649,376.139,-81.809,-176.126,9.143,148.725
C07085=1164.645,376.386,-81.844,-176.125,9.147,148.726
C07086=1164.642,376.634,-81.880,-176.123,9.150,148.727
C07087=1164.638,376.881,-81.915,-176.122,9.154,148.727
C07088=1164.634,377.129,-81.951,-176.121,9.157,148.728
C07089=1164.630,377.377,-81.987,-176.119,9.161,148.729
C07090=1164.626,377.623,-82.022,-176.118,9.165,148.729
C07091=1164.622,377.871,-82.058,-176.117,9.169,148.730
C07092=1164.618,378.118,-82.093,-176.115,9.173,148.730
C07093=1164.614,378.366,-82.130,-176.114,9.176,148.731
C07094=1164.610,378.614,-82.165,-176.113,9.180,148.732
C07095=1164.606,378.860,-82.200,-176.112,9.184,148.732
C07096=1164.603,379.107,-82.237,-176.111,9.187,148.733
C07097=1164.598,379.355,-82.273,-176.110,9.191,148.734
C07098=1164.595,379.603,-82.308,-176.108,9.195,148.734
C07099=1164.591,379.850,-82.344,-176.108,9.199,148.735
C07100=1164.586,380.098,-82.380,-176.106,9.202,148.736
C07101=1164.583,380.345,-82.415,-176.105,9.206,148.736
C07102=1164.579,380.592,-82.451,-176.104,9.210,148.737
C07103=1164.575,380.839,-82.487,-176.104,9.213,148.738
C07104=1164.571,381.087,-82.523,-176.103,9.217,148.738
C07105=1164.567,381.334,-82.559,-176.102,9.220,148.739
C07106=1164.563,381.582,-82.594,-176.101,9.224,148.740
C07107=1164.559,381.830,-82.630,-176.100,9.227,148.740
C07108=1164.556,382.077,-82.667,-176.099,9.231,148.741
C07109=1164.552,382.324,-82.702,-176.098,9.235,148.742
C07110=1164.548,382.572,-82.738,-176.098,9.238,148.743
C07111=1164.543,382.819,-82.773,-176.097,9.242,148.743
C07112=1164.540,383.066,-82.810,-176.096,9.245,148.744
C07113=1164.536,383.313,-82.846,-176.095,9.249,148.745
C07114=1164.532,383.561,-82.881,-176.095,9.252,148.746
C07115=1164.528,383.808,-82.918,-176.094,9.255,148.746
C07116=1164.524,384.056,-82.954,-176.094,9.259,148.747
C07117=1164.521,384.303,-82.989,-176.093,9.262,148.748
C07118=1164.516,384.551,-83.025,-176.093,9.265,148.748
C07119=1164.513,384.798,-83.062,-176.092,9.270,148.749
C07120=1164.508,385.046,-83.098,-176.091,9.273,148.750
C07121=1164.505,385.293,-83.133,-176.091,9.276,148.751
C07122=1164.501,385.539,-83.169,-176.091,9.279,148.751
C07123=1164.496,385.787,-83.205,-176.090,9.282,148.752
C07124=1164.493,386.035,-83.241,-176.090,9.285,148.753
C07125=1164.489,386.282,-83.278,-176.089,9.289,148.754
C07126=1164.485,386.529,-83.313,-176.089,9.292,148.754
C07127=1164.482,386.776,-83.350,-176.089,9.296,148.755
C07128=1164.477,387.024,-83.386,-176.089,9.299,148.756
C07129=1164.473,387.272,-83.421,-176.088,9.302,148.757
C07130=1164.469,387.519,-83.458,-176.088,9.305,148.758
C07131=1164.466,387.766,-83.494,-176.088,9.309,148.758
C07132=1164.462,388.013,-83.531,-176.088,9.311,148.759
C07133=1164.458,388.261,-83.566,-176.087,9.315,148.760
C07134=1164.454,388.508,-83.602,-176.087,9.317,148.761
C07135=1164.450,388.756,-83.639,-176.087,9.321,148.762
C07136=1164.447,389.003,-83.674,-176.088,9.323,148.762
C07137=1164.442,389.250,-83.711,-176.087,9.327,148.763
C07138=1164.439,389.498,-83.747,-176.087,9.329,148.764
C07139=1164.435,389.745,-83.783,-176.087,9.333,148.765
C07140=1164.431,389.992,-83.819,-176.087,9.336,148.765
C07141=1164.427,390.240,-83.856,-176.088,9.338,148.766
C07142=1164.423,390.487,-83.891,-176.087,9.342,148.767
C07143=1164.419,390.734,-83.928,-176.088,9.345,148.768
C07144=1164.416,390.982,-83.964,-176.088,9.347,148.768
C07145=1164.411,391.267,-84.005,-176.088,9.351,148.769
C07146=1164.406,391.552,-84.047,-176.088,9.353,148.770
C07147=1164.402,391.838,-84.089,-176.088,9.357,148.771
C07148=1164.398,392.123,-84.131,-176.089,9.360,148.772
C07149=1164.393,392.371,-84.167,-176.089,9.362,148.773
C07150=1164.389,392.617,-84.203,-176.089,9.365,148.774
C07151=1164.385,392.865,-84.239,-176.089,9.368,148.774
C07152=1164.382,393.112,-84.275,-176.090,9.370,148.775
C07153=1164.377,393.360,-84.312,-176.090,9.373,148.776
C07154=1164.374,393.607,-84.348,-176.090,9.376,148.777
C07155=1164.370,393.855,-84.384,-176.090,9.378,148.777
C07156=1164.367,394.102,-84.421,-176.091,9.381,148.778
C07157=1164.362,394.348,-84.457,-176.091,9.384,148.779
C07158=1164.358,394.596,-84.493,-176.091,9.387,148.780
C07159=1164.354,394.843,-84.530,-176.092,9.389,148.781
C07160=1164.351,395.091,-84.565,-176.092,9.392,148.781
C07161=1164.346,395.338,-84.602,-176.092,9.395,148.782
C07162=1164.343,395.585,-84.637,-176.093,9.397,148.783
C07163=1164.339,395.832,-84.674,-176.093,9.399,148.784
C07164=1164.335,396.080,-84.710,-176.093,9.402,148.784
C07165=1164.331,396.327,-84.747,-176.094,9.405,148.785
C07166=1164.328,396.575,-84.783,-176.094,9.407,148.786
C07167=1164.324,396.823,-84.819,-176.095,9.409,148.787
C07168=1164.320,397.070,-84.856,-176.095,9.411,148.787
C07169=1164.316,397.317,-84.892,-176.096,9.414,148.788
C07170=1164.312,397.564,-84.929,-176.096,9.416,148.789
C07171=1164.308,397.812,-84.964,-176.096,9.419,148.790
C07172=1164.304,398.059,-85.001,-176.097,9.422,148.790
C07173=1164.301,398.306,-85.037,-176.098,9.423,148.791
C07174=1164.296,398.554,-85.074,-176.098,9.426,148.792
C07175=1164.293,398.801,-85.110,-176.099,9.428,148.792
C07176=1164.289,399.049,-85.146,-176.099,9.430,148.793
C07177=1164.285,399.296,-85.183,-176.100,9.432,148.794
C07178=1164.281,399.543,-85.219,-176.100,9.435,148.795
C07179=1164.277,399.790,-85.255,-176.100,9.437,148.795
C07180=1164.273,400.037,-85.292,-176.101,9.439,148.796
C07181=1164.269,400.285,-85.328,-176.101,9.442,148.797
C07182=1164.266,400.532,-85.364,-176.102,9.444,148.798
C07183=1164.262,400.779,-85.401,-176.103,9.445,148.798
C07184=1164.257,401.027,-85.437,-176.103,9.448,148.799
C07185=1164.254,401.274,-85.473,-176.104,9.450,148.800
C07186=1164.249,401.522,-85.509,-176.104,9.452,148.800
C07187=1164.246,401.769,-85.546,-176.105,9.454,148.801
C07188=1164.242,402.016,-85.582,-176.105,9.457,148.802
C07189=1164.238,402.263,-85.618,-176.106,9.459,148.803
C07190=1164.234,402.510,-85.655,-176.106,9.460,148.803
C07191=1164.230,402.758,-85.692,-176.107,9.463,148.804
C07192=1164.227,403.005,-85.727,-176.107,9.465,148.805
C07193=1164.222,403.252,-85.764,-176.107,9.467,148.805
C07194=1164.219,403.500,-85.800,-176.108,9.469,148.806
C07195=1164.215,403.747,-85.837,-176.109,9.471,148.807
C07196=1164.211,403.994,-85.873,-176.109,9.473,148.807
C07197=1164.207,404.242,-85.909,-176.110,9.475,148.808
C07198=1164.203,404.489,-85.946,-176.110,9.477,148.809
C07199=1164.199,404.736,-85.982,-176.111,9.479,148.809
C07200=1164.195,404.984,-86.018,-176.111,9.481,148.810
C07201=1164.191,405.231,-86.055,-176.112,9.483,148.811
C07202=1164.188,405.478,-86.091,-176.113,9.485,148.811
C07203=1164.183,405.725,-86.127,-176.113,9.487,148.812
C07204=1164.180,405.973,-86.164,-176.113,9.489,148.813
C07205=1164.176,406.220,-86.201,-176.114,9.491,148.813
C07206=1164.172,406.468,-86.237,-176.115,9.493,148.814
C07207=1164.169,406.715,-86.273,-176.115,9.495,148.815
C07208=1164.165,406.962,-86.310,-176.116,9.497,148.815
C07209=1164.161,407.210,-86.346,-176.116,9.499,148.816
C07210=1164.157,407.457,-86.383,-176.117,9.500,148.817
C07211=1164.153,407.704,-86.419,-176.117,9.503,148.817
C07212=1164.149,407.951,-86.455,-176.118,9.504,148.818
C07213=1164.145,408.199,-86.492,-176.118,9.506,148.818
C07214=1164.142,408.446,-86.528,-176.119,9.508,148.819
C07215=1164.137,408.693,-86.564,-176.119,9.510,148.820
C07216=1164.133,408.941,-86.601,-176.120,9.512,148.820
C07217=1164.130,409.187,-86.637,-176.120,9.514,148.821
C07218=1164.125,409.435,-86.674,-176.121,9.515,148.822
C07219=1164.122,409.682,-86.710,-176.121,9.517,148.822
C07220=1164.118,409.929,-86.747,-176.122,9.520,148.823
C07221=1164.114,410.177,-86.784,-176.122,9.521,148.824
C07222=1164.110,410.424,-86.819,-176.123,9.523,148.824
C07223=1164.106,410.671,-86.856,-176.123,9.525,148.825
C07224=1164.102,410.919,-86.893,-176.124,9.526,148.825
C07225=1164.099,411.167,-86.929,-176.124,9.529,148.826
C07226=1164.095,411.414,-86.966,-176.124,9.530,148.826
C07227=1164.091,411.661,-87.002,-176.125,9.532,148.827
C07228=1164.087,411.908,-87.038,-176.126,9.534,148.828
C07229=1164.083,412.156,-87.075,-176.126,9.535,148.828
C07230=1164.080,412.403,-87.111,-176.127,9.537,148.829
C07231=1164.075,412.650,-87.148,-176.127,9.540,148.830
C07232=1164.071,412.898,-87.184,-176.127,9.541,148.830
C07233=1164.068,413.144,-87.220,-176.128,9.543,148.831
C07234=1164.064,413.392,-87.257,-176.128,9.544,148.831
C07235=1164.059,413.639,-87.293,-176.129,9.546,148.832
C07236=1164.056,413.886,-87.330,-176.129,9.548,148.832
C07237=1164.052,414.134,-87.366,-176.129,9.550,148.833
C07238=1164.048,414.380,-87.403,-176.130,9.552,148.834
C07239=1164.044,414.628,-87.439,-176.130,9.553,148.834
C07240=1164.040,414.875,-87.476,-176.131,9.555,148.835
C07241=1164.037,415.123,-87.512,-176.131,9.557,148.835
C07242=1164.033,415.370,-87.549,-176.131,9.559,148.836
C07243=1164.031,415.617,-87.585,-176.132,9.561,148.836
C07244=1164.029,415.865,-87.621,-176.132,9.562,148.837
C07245=1164.028,416.199,-87.670,-176.132,9.565,148.838
C07246=1164.029,416.531,-87.718,-176.134,9.567,148.838
C07247=1164.032,416.864,-87.767,-176.134,9.569,148.839
C07248=1164.036,417.197,-87.815,-176.134,9.571,148.840
C07249=1163.615,417.199,-87.861,-176.137,9.582,148.843
C07250=1163.610,416.862,-87.812,-176.136,9.580,148.843
C07251=1163.608,416.527,-87.764,-176.136,9.577,148.842
C07252=1163.607,416.190,-87.715,-176.136,9.576,148.841
C07253=1163.608,415.854,-87.665,-176.135,9.573,148.841
C07254=1163.610,415.606,-87.629,-176.135,9.571,148.840
C07255=1163.613,415.359,-87.593,-176.134,9.570,148.840
C07256=1163.615,415.111,-87.556,-176.134,9.568,148.839
C07257=1163.619,414.864,-87.520,-176.134,9.566,148.838
C07258=1163.623,414.617,-87.483,-176.133,9.564,148.838
C07259=1163.627,414.369,-87.447,-176.133,9.562,148.837
C07260=1163.631,414.122,-87.411,-176.132,9.561,148.837
C07261=1163.635,413.875,-87.374,-176.132,9.559,148.836
C07262=1163.639,413.628,-87.337,-176.132,9.557,148.835
C07263=1163.643,413.381,-87.301,-176.131,9.555,148.835
C07264=1163.647,413.133,-87.264,-176.131,9.553,148.834
C07265=1163.651,412.886,-87.228,-176.130,9.552,148.834
C07266=1163.654,412.639,-87.192,-176.130,9.550,148.833
C07267=1163.658,412.391,-87.155,-176.129,9.548,148.832
C07268=1163.663,412.144,-87.118,-176.129,9.546,148.832
C07269=1163.666,411.897,-87.082,-176.129,9.544,148.831
C07270=1163.670,411.650,-87.046,-176.128,9.543,148.831
C07271=1163.674,411.402,-87.009,-176.127,9.541,148.830
C07272=1163.677,411.155,-86.972,-176.127,9.540,148.830
C07273=1163.682,410.907,-86.936,-176.127,9.537,148.829
C07274=1163.685,410.660,-86.900,-176.126,9.535,148.828
C07275=1163.689,410.413,-86.863,-176.126,9.534,148.828
C07276=1163.693,410.166,-86.826,-176.125,9.532,148.827
C07277=1163.697,409.918,-86.791,-176.124,9.530,148.826
C07278=1163.701,409.671,-86.754,-176.124,9.529,148.826
C07279=1163.705,409.424,-86.717,-176.124,9.526,148.825
C07280=1163.709,409.176,-86.682,-176.123,9.525,148.825
C07281=1163.713,408.929,-86.645,-176.123,9.523,148.824
C07282=1163.716,408.682,-86.608,-176.122,9.521,148.823
C07283=1163.720,408.434,-86.572,-176.121,9.519,148.823
C07284=1163.725,408.187,-86.535,-176.121,9.517,148.822
C07285=1163.728,407.940,-86.499,-176.120,9.515,148.821
C07286=1163.732,407.693,-86.463,-176.120,9.514,148.821
C07287=1163.736,407.446,-86.427,-176.119,9.512,148.820
C07288=1163.740,407.199,-86.390,-176.119,9.509,148.820
C07289=1163.743,406.951,-86.353,-176.118,9.508,148.819
C07290=1163.747,406.703,-86.317,-176.118,9.506,148.818
C07291=1163.751,406.456,-86.280,-176.117,9.504,148.818
C07292=1163.755,406.209,-86.243,-176.116,9.502,148.817
C07293=1163.759,405.961,-86.208,-176.116,9.500,148.816
C07294=1163.763,405.714,-86.171,-176.116,9.498,148.816
C07295=1163.766,405.467,-86.135,-176.115,9.496,148.815
C07296=1163.771,405.219,-86.099,-176.115,9.494,148.814
C07297=1163.775,404.972,-86.062,-176.114,9.492,148.814
C07298=1163.778,404.725,-86.025,-176.113,9.490,148.813
C07299=1163.782,404.477,-85.989,-176.113,9.488,148.812
C07300=1163.786,404.231,-85.953,-176.112,9.486,148.812
C07301=1163.790,403.983,-85.916,-176.112,9.484,148.811
C07302=1163.794,403.736,-85.880,-176.111,9.482,148.810
C07303=1163.798,403.489,-85.844,-176.111,9.480,148.810
C07304=1163.802,403.242,-85.807,-176.110,9.478,148.809
C07305=1163.805,402.994,-85.771,-176.110,9.476,148.808
C07306=1163.810,402.747,-85.735,-176.109,9.474,148.808
C07307=1163.814,402.499,-85.698,-176.109,9.472,148.807
C07308=1163.817,402.252,-85.662,-176.108,9.470,148.806
C07309=1163.821,402.005,-85.625,-176.107,9.467,148.805
C07310=1163.825,401.757,-85.590,-176.107,9.466,148.805
C07311=1163.829,401.510,-85.553,-176.107,9.463,148.804
C07312=1163.832,401.263,-85.516,-176.106,9.461,148.803
C07313=1163.836,401.015,-85.480,-176.105,9.460,148.803
C07314=1163.840,400.768,-85.443,-176.105,9.457,148.802
C07315=1163.844,400.521,-85.407,-176.104,9.455,148.801
C07316=1163.848,400.273,-85.371,-176.104,9.452,148.800
C07317=1163.852,400.026,-85.335,-176.103,9.451,148.800
C07318=1163.856,399.778,-85.298,-176.103,9.448,148.799
C07319=1163.860,399.531,-85.262,-176.102,9.446,148.798
C07320=1163.863,399.284,-85.225,-176.102,9.443,148.797
C07321=1163.868,399.036,-85.189,-176.101,9.442,148.797
C07322=1163.871,398.790,-85.153,-176.101,9.439,148.796
C07323=1163.875,398.542,-85.116,-176.100,9.437,148.795
C07324=1163.879,398.295,-85.080,-176.100,9.434,148.795
